// TwinCAT 3 PLC project plc_tmo_hutch_vac
// ProgramVersion: 3.1.4022.7
// libraries:
//   LCLS General, * (SLAC)
//   LCLS Vacuum, * (SLAC - LCLS)
//   LCLSVacuumSerialDriverLib, * (SLAC - LCLS)
//   PMPS, * (SLAC - LCLS)
//   Tc2_SerialCom, * (Beckhoff Automation GmbH)
//   Tc2_Standard, * (Beckhoff Automation GmbH)
//   Tc2_System, * (Beckhoff Automation GmbH)
//   Tc3_Module, * (Beckhoff Automation GmbH)
// project tree:
//   / ComTask.TcTTO, FSVTask.TcTTO, PlcTask.TcTTO
//   GVLs/ GVL_COM.TcGVL (not stored), GVL_FSV_PMPS.TcGVL (not stored), GVL_FS_Devices.TcGVL (not stored), GVL_Hutch_Gauges.TcGVL, GVL_Hutch_Pumps.TcGVL, GVL_Hutch_Valves.TcGVL, GVL_PMPS.TcGVL (not stored), GVL_Variables.TcGVL
//   POUs/ F_Turbo_Protection_ILK.TcPOU, MAIN.TcPOU, PMPS.TcPOU (not stored), PRG_COM.TcPOU (not stored), PRG_FEE.TcPOU, PRG_FSV.TcPOU (not stored), PRG_Hutch_Beamline_Valves.TcPOU, PRG_Hutch_Gauges.TcPOU, PRG_Roughing_Pumps.TcPOU
// real-time tasks:
//   TASK PlcTask: cycle T#10ms, priority 20, ADS port 350
//   TASK ComTask: cycle T#12ms, priority 21, ADS port 351
//   TASK FSVTask: cycle T#2ms, priority 19, ADS port 352
// I/O:
//   DEVICE Device 1 (EtherCAT), AmsNetId 172.21.132.45.2.1
//     Term 1 (EK1200)
//     TMO_WALL_WEST_EP01 (EP4374-0002)
//     TMO_K4S2_DRL_01 (EK1100) [EK1100 EtherCAT Coupler (2A E-Bus)]
//       K4S2_01_E1_VFS (EL1004)
//       K4S2_01_E2 (EL9190) [EL9190 Power Supplier]
//       K4S2_01_E3_VFS (EL2202)
//       K4S2_01_E4_VFS (EL2202)
//       K4S2_01_E5 (EL1004)
//       K4S2_01_E6 (EL2004)
//       Term 31 (EL9011)
//     TMO_K4S2_DRL_02 (EK1100) [EK1100 EtherCAT Coupler (2A E-Bus)]
//       K4S2_02_E1 (EL3174)
//       K4S2_02_E2 (EL3174)
//       K4S2_02_E3 (EL9184)
//       K4S2_02_E4 (EL9070) [EL9070 Shield terminal]
//       K4S2_02_E5 (EL2624)
//       K4S2_02_E6 (EL9505)
//       K4S2_02_E7 (EL1124) [EL1124 4Ch. Dig. Input 5V, 10µs, Sensor Power]
//       K4S2_02_E8 (EL1124)
//       K4S2_02_E9 (EL9410)
//       K4S2_02_E10 (EL6021) [EL6021 Interface (RS422/485)]
//       K4S2_02_E11 (EL1004)
//       K4S2_02_E12 (EL2794)
//       K4S2_02_E13 (EL1004)
//       K4S2_02_E14 (EL2794)
//       K4S2_02_E15 (EL1004)
//       K4S2_02_E16 (EL2794)
//       K4S2_02_E17 (EL6001) [EL6001 Interface (RS232)]
//       K4S2_02_E18 (EL6001) [EL6001 Interface (RS232)]
//       K4S2_02_E19 (EL1004)
//       K4S2_02_E20 (EL2004)
//       Term 32 (EL9011)
//     TMO_K4S2_ EP1 (EP4374-0002) [EP4374-0002 2Ch. Ana. Input +/-10V, 0-10V, 0/4-20mA configurable; 2Ch. Ana. Output +/-10V, 0-10V, 0/4-20mA configurable]
//     TMO_K4S6_ EP1 (EP4374-0002) [EP4374-0002 2Ch. Ana. Input +/-10V, 0-10V, 0/4-20mA configurable; 2Ch. Ana. Output +/-10V, 0-10V, 0/4-20mA configurable]
//     TMO_K4S6_DRL_01 (EK1100) [EK1100 EtherCAT Coupler (2A E-Bus)]
//       K4S6_01_E1 (EL1004)
//       K4S6_01_E2 (EL2004)
//       K4S6_01_E3 (EL1004)
//       K4S6_01_E4 (EL2004)
//       K4S6_01_E5 (EL6021) [EL6021 Schnittstelle (RS422/485)]
//       K4S6_01_E6 (EL1004)
//       K4S6_01_E7 (EL2004)
//       K4S6_01_E8 (EL1004)
//       K4S6_01_E9 (EL2004)
//       K4S6_01_E10 (EL6021)
//       K4S6_01_E11 (EL1004)
//       K4S6_01_E12 (EL2004)
//       K4S6_01_E13 (EL9410)
//       K4S6_01_E14 (EL2624)
//       K4S6_01_E15 (EL3174)
//       K4S6_01_E16 (EL9184) [EL9184 Potential Connection, 8 x 24V, 8 x Ground]
//       K4S6_01_E17 (EL9070) [EL9070 Shield terminal]
//       K4S6_01_E18 (EL3174)
//       K4S6_01_E19 (EL9505)
//       K4S6_01_E20 (EL1124)
//       K4S6_01_E21 (EL1124)
//       Term 119 (EL9410)
//       K4S6_01_E22_IP1 (EL1004)
//       K4S6_01_E23_IP1 (EL2794)
//       Term 91 (EL9011)
//     TMO_K4S8_DRL_01 (EK1100) [EK1100 EtherCAT Coupler (2A E-Bus)]
//       K4S8_01_E1 (EL1004)
//       K4S8_01_E2 (EL9190) [EL9190 Power Supplier]
//       K4S8_01_E3 (EL2202)
//       K4S8_01_E4 (EL2202)
//       K4S8_01_E5 (EL1004)
//       K4S8_01_E6 (EL2004)
//       Term 92 (EL9011)
// variable links:
//   plc_tmo_hutch_vac_fs/plc_tmo_hutch_vac_fs Instance <-> Device 1 (EtherCAT)/TMO_K4S2_DRL_01 (EK1100)/K4S2_01_E1_VFS (EL1004)
//     PlcTask Inputs/GVL_FS_Devices.MR3K4_KBO_VFS_1.i_xClsLS <-> Channel 1/Input
//     PlcTask Inputs/GVL_FS_Devices.MR3K4_KBO_VFS_1.i_xOpnLS <-> Channel 2/Input
//   plc_tmo_hutch_vac_fs/plc_tmo_hutch_vac_fs Instance <-> Device 1 (EtherCAT)/TMO_K4S2_DRL_01 (EK1100)/K4S2_01_E3_VFS (EL2202)
//     PlcTask Outputs/GVL_FS_Devices.MR3K4_KBO_VFS_1.q_xClose_A <-> Channel 1/Output
//     PlcTask Outputs/GVL_FS_Devices.MR3K4_KBO_VFS_1.q_xClose_B <-> Channel 2/Output
//   plc_tmo_hutch_vac_fs/plc_tmo_hutch_vac_fs Instance <-> Device 1 (EtherCAT)/TMO_K4S2_DRL_01 (EK1100)/K4S2_01_E4_VFS (EL2202)
//     PlcTask Outputs/GVL_FS_Devices.MR3K4_KBO_VFS_1.q_xClose_C <-> Channel 1/Output
//     PlcTask Outputs/GVL_FS_Devices.MR3K4_KBO_VFS_1.q_xOPN_DO <-> Channel 2/Output
//   plc_tmo_hutch_vac_fs/plc_tmo_hutch_vac_fs Instance <-> Device 1 (EtherCAT)/TMO_K4S8_DRL_01 (EK1100)/K4S8_01_E1 (EL1004)
//     PlcTask Inputs/GVL_FS_Devices.MR4K4_KBO_VFS_1.i_xClsLS <-> Channel 1/Input
//     PlcTask Inputs/GVL_FS_Devices.MR4K4_KBO_VFS_1.i_xOpnLS <-> Channel 2/Input
//   plc_tmo_hutch_vac_fs/plc_tmo_hutch_vac_fs Instance <-> Device 1 (EtherCAT)/TMO_K4S8_DRL_01 (EK1100)/K4S8_01_E3 (EL2202)
//     PlcTask Outputs/GVL_FS_Devices.MR4K4_KBO_VFS_1.q_xClose_A <-> Channel 1/Output
//     PlcTask Outputs/GVL_FS_Devices.MR4K4_KBO_VFS_1.q_xClose_B <-> Channel 2/Output
//   plc_tmo_hutch_vac_fs/plc_tmo_hutch_vac_fs Instance <-> Device 1 (EtherCAT)/TMO_K4S8_DRL_01 (EK1100)/K4S8_01_E4 (EL2202)
//     PlcTask Outputs/GVL_FS_Devices.MR4K4_KBO_VFS_1.q_xClose_C <-> Channel 1/Output
//     PlcTask Outputs/GVL_FS_Devices.MR4K4_KBO_VFS_1.q_xOPN_DO <-> Channel 2/Output
//   plc_tmo_hutch_vac Instance <-> Device 1 (EtherCAT)/TMO_K4S2_ EP1 (EP4374-0002)
//     ComTask Outputs/GVL_Hutch_Valves.TMO_ROUGH1_VFV_02.q_iRawPosition <-> AO Outputs Channel 3/Analog output
//     ComTask Outputs/GVL_Hutch_Valves.TMO_ROUGH2_VFV_01.q_iRawPosition <-> AO Outputs Channel 4/Analog output
//     PlcTask Inputs/GVL_Hutch_Gauges.TMO_ROUGH1_GPI_02.i_iPRESS_R <-> AI Inputs Channel 1/Value
//     PlcTask Inputs/GVL_Hutch_Gauges.TMO_ROUGH2_GPI_02.i_iPRESS_R <-> AI Inputs Channel 2/Value
//   plc_tmo_hutch_vac Instance <-> Device 1 (EtherCAT)/TMO_K4S2_DRL_01 (EK1100)/K4S2_01_E1_VFS (EL1004)
//     FSVTask Inputs/GVL_FS_Devices.MR3K4_KBO_VFS_1.i_xClsLS <-> Channel 1/Input
//     FSVTask Inputs/GVL_FS_Devices.MR3K4_KBO_VFS_1.i_xOpnLS <-> Channel 2/Input
//   plc_tmo_hutch_vac Instance <-> Device 1 (EtherCAT)/TMO_K4S2_DRL_01 (EK1100)/K4S2_01_E3_VFS (EL2202)
//     FSVTask Outputs/GVL_FS_Devices.MR3K4_KBO_VFS_1.q_xClose_A <-> Channel 1/Output
//     FSVTask Outputs/GVL_FS_Devices.MR3K4_KBO_VFS_1.q_xClose_B <-> Channel 2/Output
//   plc_tmo_hutch_vac Instance <-> Device 1 (EtherCAT)/TMO_K4S2_DRL_01 (EK1100)/K4S2_01_E4_VFS (EL2202)
//     FSVTask Outputs/GVL_FS_Devices.MR3K4_KBO_VFS_1.q_xClose_C <-> Channel 1/Output
//     FSVTask Outputs/GVL_FS_Devices.MR3K4_KBO_VFS_1.q_xOPN_DO <-> Channel 2/Output
//   plc_tmo_hutch_vac Instance <-> Device 1 (EtherCAT)/TMO_K4S2_DRL_01 (EK1100)/K4S2_01_E5 (EL1004)
//     PlcTask Inputs/GVL_Hutch_Valves.MR2K4_KBO_VWC_01.i_xClsLS <-> Channel 2/Input
//     PlcTask Inputs/GVL_Hutch_Valves.MR3K4_KBO_VWC_01.i_xClsLS <-> Channel 4/Input
//     PlcTask Inputs/GVL_Hutch_Valves.MR2K4_KBO_VWC_01.i_xOpnLS <-> Channel 1/Input
//     PlcTask Inputs/GVL_Hutch_Valves.MR3K4_KBO_VWC_01.i_xOpnLS <-> Channel 3/Input
//   plc_tmo_hutch_vac Instance <-> Device 1 (EtherCAT)/TMO_K4S2_DRL_01 (EK1100)/K4S2_01_E6 (EL2004)
//     PlcTask Outputs/GVL_Hutch_Valves.MR2K4_KBO_VWC_01.q_xOPN_DO <-> Channel 1/Output
//     PlcTask Outputs/GVL_Hutch_Valves.MR3K4_KBO_VWC_01.q_xOPN_DO <-> Channel 2/Output
//   plc_tmo_hutch_vac Instance <-> Device 1 (EtherCAT)/TMO_K4S2_DRL_02 (EK1100)/K4S2_02_E1 (EL3174)
//     PlcTask Inputs/GVL_Hutch_Gauges.MR2K4_KBO_GCC_01.i_iPRESS_R <-> AI Standard Channel 3/Value
//     PlcTask Inputs/GVL_Hutch_Gauges.MR2K4_KBO_GPI_01.i_iPRESS_R <-> AI Standard Channel 2/Value
//     PlcTask Inputs/GVL_Hutch_Gauges.PA1K4_IP1_GCC_01.i_iPRESS_R <-> AI Standard Channel 4/Value
//   plc_tmo_hutch_vac Instance <-> Device 1 (EtherCAT)/TMO_K4S2_DRL_02 (EK1100)/K4S2_02_E10 (EL6021)
//     ComTask Inputs/GVL_COM.K4S2_02_E10_stComIn/D[0] <-> COM TxPDO-Map Inputs/Data In 0
//     ComTask Inputs/GVL_COM.K4S2_02_E10_stComIn/D[10] <-> COM TxPDO-Map Inputs/Data In 10
//     ComTask Inputs/GVL_COM.K4S2_02_E10_stComIn/D[11] <-> COM TxPDO-Map Inputs/Data In 11
//     ComTask Inputs/GVL_COM.K4S2_02_E10_stComIn/D[12] <-> COM TxPDO-Map Inputs/Data In 12
//     ComTask Inputs/GVL_COM.K4S2_02_E10_stComIn/D[13] <-> COM TxPDO-Map Inputs/Data In 13
//     ComTask Inputs/GVL_COM.K4S2_02_E10_stComIn/D[14] <-> COM TxPDO-Map Inputs/Data In 14
//     ComTask Inputs/GVL_COM.K4S2_02_E10_stComIn/D[15] <-> COM TxPDO-Map Inputs/Data In 15
//     ComTask Inputs/GVL_COM.K4S2_02_E10_stComIn/D[16] <-> COM TxPDO-Map Inputs/Data In 16
//     ComTask Inputs/GVL_COM.K4S2_02_E10_stComIn/D[17] <-> COM TxPDO-Map Inputs/Data In 17
//     ComTask Inputs/GVL_COM.K4S2_02_E10_stComIn/D[18] <-> COM TxPDO-Map Inputs/Data In 18
//     ComTask Inputs/GVL_COM.K4S2_02_E10_stComIn/D[19] <-> COM TxPDO-Map Inputs/Data In 19
//     ComTask Inputs/GVL_COM.K4S2_02_E10_stComIn/D[1] <-> COM TxPDO-Map Inputs/Data In 1
//     ComTask Inputs/GVL_COM.K4S2_02_E10_stComIn/D[20] <-> COM TxPDO-Map Inputs/Data In 20
//     ComTask Inputs/GVL_COM.K4S2_02_E10_stComIn/D[21] <-> COM TxPDO-Map Inputs/Data In 21
//     ComTask Inputs/GVL_COM.K4S2_02_E10_stComIn/D[2] <-> COM TxPDO-Map Inputs/Data In 2
//     ComTask Inputs/GVL_COM.K4S2_02_E10_stComIn/D[3] <-> COM TxPDO-Map Inputs/Data In 3
//     ComTask Inputs/GVL_COM.K4S2_02_E10_stComIn/D[4] <-> COM TxPDO-Map Inputs/Data In 4
//     ComTask Inputs/GVL_COM.K4S2_02_E10_stComIn/D[5] <-> COM TxPDO-Map Inputs/Data In 5
//     ComTask Inputs/GVL_COM.K4S2_02_E10_stComIn/D[6] <-> COM TxPDO-Map Inputs/Data In 6
//     ComTask Inputs/GVL_COM.K4S2_02_E10_stComIn/D[7] <-> COM TxPDO-Map Inputs/Data In 7
//     ComTask Inputs/GVL_COM.K4S2_02_E10_stComIn/D[8] <-> COM TxPDO-Map Inputs/Data In 8
//     ComTask Inputs/GVL_COM.K4S2_02_E10_stComIn/D[9] <-> COM TxPDO-Map Inputs/Data In 9
//     ComTask Inputs/GVL_COM.K4S2_02_E10_stComIn/Status <-> COM TxPDO-Map Inputs/Status
//     ComTask Outputs/GVL_COM.K4S2_02_E10_stComOut/Ctrl <-> COM RxPDO-Map Outputs/Ctrl
//     ComTask Outputs/GVL_COM.K4S2_02_E10_stComOut/D[0] <-> COM RxPDO-Map Outputs/Data Out 0
//     ComTask Outputs/GVL_COM.K4S2_02_E10_stComOut/D[10] <-> COM RxPDO-Map Outputs/Data Out 10
//     ComTask Outputs/GVL_COM.K4S2_02_E10_stComOut/D[11] <-> COM RxPDO-Map Outputs/Data Out 11
//     ComTask Outputs/GVL_COM.K4S2_02_E10_stComOut/D[12] <-> COM RxPDO-Map Outputs/Data Out 12
//     ComTask Outputs/GVL_COM.K4S2_02_E10_stComOut/D[13] <-> COM RxPDO-Map Outputs/Data Out 13
//     ComTask Outputs/GVL_COM.K4S2_02_E10_stComOut/D[14] <-> COM RxPDO-Map Outputs/Data Out 14
//     ComTask Outputs/GVL_COM.K4S2_02_E10_stComOut/D[15] <-> COM RxPDO-Map Outputs/Data Out 15
//     ComTask Outputs/GVL_COM.K4S2_02_E10_stComOut/D[16] <-> COM RxPDO-Map Outputs/Data Out 16
//     ComTask Outputs/GVL_COM.K4S2_02_E10_stComOut/D[17] <-> COM RxPDO-Map Outputs/Data Out 17
//     ComTask Outputs/GVL_COM.K4S2_02_E10_stComOut/D[18] <-> COM RxPDO-Map Outputs/Data Out 18
//     ComTask Outputs/GVL_COM.K4S2_02_E10_stComOut/D[19] <-> COM RxPDO-Map Outputs/Data Out 19
//     ComTask Outputs/GVL_COM.K4S2_02_E10_stComOut/D[1] <-> COM RxPDO-Map Outputs/Data Out 1
//     ComTask Outputs/GVL_COM.K4S2_02_E10_stComOut/D[20] <-> COM RxPDO-Map Outputs/Data Out 20
//     ComTask Outputs/GVL_COM.K4S2_02_E10_stComOut/D[21] <-> COM RxPDO-Map Outputs/Data Out 21
//     ComTask Outputs/GVL_COM.K4S2_02_E10_stComOut/D[2] <-> COM RxPDO-Map Outputs/Data Out 2
//     ComTask Outputs/GVL_COM.K4S2_02_E10_stComOut/D[3] <-> COM RxPDO-Map Outputs/Data Out 3
//     ComTask Outputs/GVL_COM.K4S2_02_E10_stComOut/D[4] <-> COM RxPDO-Map Outputs/Data Out 4
//     ComTask Outputs/GVL_COM.K4S2_02_E10_stComOut/D[5] <-> COM RxPDO-Map Outputs/Data Out 5
//     ComTask Outputs/GVL_COM.K4S2_02_E10_stComOut/D[6] <-> COM RxPDO-Map Outputs/Data Out 6
//     ComTask Outputs/GVL_COM.K4S2_02_E10_stComOut/D[7] <-> COM RxPDO-Map Outputs/Data Out 7
//     ComTask Outputs/GVL_COM.K4S2_02_E10_stComOut/D[8] <-> COM RxPDO-Map Outputs/Data Out 8
//     ComTask Outputs/GVL_COM.K4S2_02_E10_stComOut/D[9] <-> COM RxPDO-Map Outputs/Data Out 9
//   plc_tmo_hutch_vac Instance <-> Device 1 (EtherCAT)/TMO_K4S2_DRL_02 (EK1100)/K4S2_02_E11 (EL1004)
//     PlcTask Inputs/GVL_Hutch_Pumps.PA1K4_IP1_PTM_01.i_xAtSpd <-> Channel 2/Input
//     PlcTask Inputs/GVL_Hutch_Pumps.PA1K4_IP1_PTM_02.i_xAtSpd <-> Channel 4/Input
//     PlcTask Inputs/GVL_Hutch_Pumps.PA1K4_IP1_PTM_01.i_xFaultNC <-> Channel 1/Input
//     PlcTask Inputs/GVL_Hutch_Pumps.PA1K4_IP1_PTM_02.i_xFaultNC <-> Channel 3/Input
//   plc_tmo_hutch_vac Instance <-> Device 1 (EtherCAT)/TMO_K4S2_DRL_02 (EK1100)/K4S2_02_E12 (EL2794)
//     PlcTask Outputs/GVL_Hutch_Pumps.PA1K4_IP1_PTM_01.q_RunDO <-> Channel 1/Output
//     PlcTask Outputs/GVL_Hutch_Pumps.PA1K4_IP1_PTM_02.q_RunDO <-> Channel 3/Output
//     PlcTask Outputs/GVL_Hutch_Pumps.PA1K4_IP1_PTM_01.q_xReset <-> Channel 2/Output
//     PlcTask Outputs/GVL_Hutch_Pumps.PA1K4_IP1_PTM_02.q_xReset <-> Channel 4/Output
//   plc_tmo_hutch_vac Instance <-> Device 1 (EtherCAT)/TMO_K4S2_DRL_02 (EK1100)/K4S2_02_E13 (EL1004)
//     PlcTask Inputs/GVL_Hutch_Pumps.PA1K4_IP1_PTM_03.i_xAtSpd <-> Channel 2/Input
//     PlcTask Inputs/GVL_Hutch_Pumps.PA1K4_IP1_PTM_03.i_xFaultNC <-> Channel 1/Input
//   plc_tmo_hutch_vac Instance <-> Device 1 (EtherCAT)/TMO_K4S2_DRL_02 (EK1100)/K4S2_02_E14 (EL2794)
//     PlcTask Outputs/GVL_Hutch_Pumps.PA1K4_IP1_PTM_03.q_RunDO <-> Channel 1/Output
//     PlcTask Outputs/GVL_Hutch_Pumps.PA1K4_IP1_PTM_03.q_xReset <-> Channel 2/Output
//   plc_tmo_hutch_vac Instance <-> Device 1 (EtherCAT)/TMO_K4S2_DRL_02 (EK1100)/K4S2_02_E15 (EL1004)
//     PlcTask Inputs/GVL_Hutch_Pumps.IM4K4_PPM_PTM_01.i_xAtSpd <-> Channel 2/Input
//     PlcTask Inputs/GVL_Hutch_Pumps.IM4K4_PPM_PTM_01.i_xFaultNC <-> Channel 1/Input
//     PlcTask Inputs/GVL_Hutch_Pumps.LI1K4_IP1_PTM_01.i_xAtSpd <-> Channel 4/Input
//     PlcTask Inputs/GVL_Hutch_Pumps.LI1K4_IP1_PTM_01.i_xFaultNC <-> Channel 3/Input
//   plc_tmo_hutch_vac Instance <-> Device 1 (EtherCAT)/TMO_K4S2_DRL_02 (EK1100)/K4S2_02_E16 (EL2794)
//     PlcTask Outputs/GVL_Hutch_Pumps.IM4K4_PPM_PTM_01.q_RunDO <-> Channel 1/Output
//     PlcTask Outputs/GVL_Hutch_Pumps.LI1K4_IP1_PTM_01.q_RunDO <-> Channel 2/Output
//   plc_tmo_hutch_vac Instance <-> Device 1 (EtherCAT)/TMO_K4S2_DRL_02 (EK1100)/K4S2_02_E17 (EL6001)
//     ComTask Inputs/GVL_COM.K4S2_02_E17_stComIn/D[0] <-> COM Inputs/Data In 0
//     ComTask Inputs/GVL_COM.K4S2_02_E17_stComIn/D[10] <-> COM Inputs/Data In 10
//     ComTask Inputs/GVL_COM.K4S2_02_E17_stComIn/D[11] <-> COM Inputs/Data In 11
//     ComTask Inputs/GVL_COM.K4S2_02_E17_stComIn/D[12] <-> COM Inputs/Data In 12
//     ComTask Inputs/GVL_COM.K4S2_02_E17_stComIn/D[13] <-> COM Inputs/Data In 13
//     ComTask Inputs/GVL_COM.K4S2_02_E17_stComIn/D[14] <-> COM Inputs/Data In 14
//     ComTask Inputs/GVL_COM.K4S2_02_E17_stComIn/D[15] <-> COM Inputs/Data In 15
//     ComTask Inputs/GVL_COM.K4S2_02_E17_stComIn/D[16] <-> COM Inputs/Data In 16
//     ComTask Inputs/GVL_COM.K4S2_02_E17_stComIn/D[17] <-> COM Inputs/Data In 17
//     ComTask Inputs/GVL_COM.K4S2_02_E17_stComIn/D[18] <-> COM Inputs/Data In 18
//     ComTask Inputs/GVL_COM.K4S2_02_E17_stComIn/D[19] <-> COM Inputs/Data In 19
//     ComTask Inputs/GVL_COM.K4S2_02_E17_stComIn/D[1] <-> COM Inputs/Data In 1
//     ComTask Inputs/GVL_COM.K4S2_02_E17_stComIn/D[20] <-> COM Inputs/Data In 20
//     ComTask Inputs/GVL_COM.K4S2_02_E17_stComIn/D[21] <-> COM Inputs/Data In 21
//     ComTask Inputs/GVL_COM.K4S2_02_E17_stComIn/D[2] <-> COM Inputs/Data In 2
//     ComTask Inputs/GVL_COM.K4S2_02_E17_stComIn/D[3] <-> COM Inputs/Data In 3
//     ComTask Inputs/GVL_COM.K4S2_02_E17_stComIn/D[4] <-> COM Inputs/Data In 4
//     ComTask Inputs/GVL_COM.K4S2_02_E17_stComIn/D[5] <-> COM Inputs/Data In 5
//     ComTask Inputs/GVL_COM.K4S2_02_E17_stComIn/D[6] <-> COM Inputs/Data In 6
//     ComTask Inputs/GVL_COM.K4S2_02_E17_stComIn/D[7] <-> COM Inputs/Data In 7
//     ComTask Inputs/GVL_COM.K4S2_02_E17_stComIn/D[8] <-> COM Inputs/Data In 8
//     ComTask Inputs/GVL_COM.K4S2_02_E17_stComIn/D[9] <-> COM Inputs/Data In 9
//     ComTask Inputs/GVL_COM.K4S2_02_E17_stComIn/Status <-> COM Inputs/Status
//     ComTask Outputs/GVL_COM.K4S2_02_E17_stComOut/Ctrl <-> COM Outputs/Ctrl
//     ComTask Outputs/GVL_COM.K4S2_02_E17_stComOut/D[0] <-> COM Outputs/Data Out 0
//     ComTask Outputs/GVL_COM.K4S2_02_E17_stComOut/D[10] <-> COM Outputs/Data Out 10
//     ComTask Outputs/GVL_COM.K4S2_02_E17_stComOut/D[11] <-> COM Outputs/Data Out 11
//     ComTask Outputs/GVL_COM.K4S2_02_E17_stComOut/D[12] <-> COM Outputs/Data Out 12
//     ComTask Outputs/GVL_COM.K4S2_02_E17_stComOut/D[13] <-> COM Outputs/Data Out 13
//     ComTask Outputs/GVL_COM.K4S2_02_E17_stComOut/D[14] <-> COM Outputs/Data Out 14
//     ComTask Outputs/GVL_COM.K4S2_02_E17_stComOut/D[15] <-> COM Outputs/Data Out 15
//     ComTask Outputs/GVL_COM.K4S2_02_E17_stComOut/D[16] <-> COM Outputs/Data Out 16
//     ComTask Outputs/GVL_COM.K4S2_02_E17_stComOut/D[17] <-> COM Outputs/Data Out 17
//     ComTask Outputs/GVL_COM.K4S2_02_E17_stComOut/D[18] <-> COM Outputs/Data Out 18
//     ComTask Outputs/GVL_COM.K4S2_02_E17_stComOut/D[19] <-> COM Outputs/Data Out 19
//     ComTask Outputs/GVL_COM.K4S2_02_E17_stComOut/D[1] <-> COM Outputs/Data Out 1
//     ComTask Outputs/GVL_COM.K4S2_02_E17_stComOut/D[20] <-> COM Outputs/Data Out 20
//     ComTask Outputs/GVL_COM.K4S2_02_E17_stComOut/D[21] <-> COM Outputs/Data Out 21
//     ComTask Outputs/GVL_COM.K4S2_02_E17_stComOut/D[2] <-> COM Outputs/Data Out 2
//     ComTask Outputs/GVL_COM.K4S2_02_E17_stComOut/D[3] <-> COM Outputs/Data Out 3
//     ComTask Outputs/GVL_COM.K4S2_02_E17_stComOut/D[4] <-> COM Outputs/Data Out 4
//     ComTask Outputs/GVL_COM.K4S2_02_E17_stComOut/D[5] <-> COM Outputs/Data Out 5
//     ComTask Outputs/GVL_COM.K4S2_02_E17_stComOut/D[6] <-> COM Outputs/Data Out 6
//     ComTask Outputs/GVL_COM.K4S2_02_E17_stComOut/D[7] <-> COM Outputs/Data Out 7
//     ComTask Outputs/GVL_COM.K4S2_02_E17_stComOut/D[8] <-> COM Outputs/Data Out 8
//     ComTask Outputs/GVL_COM.K4S2_02_E17_stComOut/D[9] <-> COM Outputs/Data Out 9
//   plc_tmo_hutch_vac Instance <-> Device 1 (EtherCAT)/TMO_K4S2_DRL_02 (EK1100)/K4S2_02_E18 (EL6001)
//     ComTask Inputs/GVL_COM.K4S2_02_E18_stComIn/D[0] <-> COM Inputs/Data In 0
//     ComTask Inputs/GVL_COM.K4S2_02_E18_stComIn/D[10] <-> COM Inputs/Data In 10
//     ComTask Inputs/GVL_COM.K4S2_02_E18_stComIn/D[11] <-> COM Inputs/Data In 11
//     ComTask Inputs/GVL_COM.K4S2_02_E18_stComIn/D[12] <-> COM Inputs/Data In 12
//     ComTask Inputs/GVL_COM.K4S2_02_E18_stComIn/D[13] <-> COM Inputs/Data In 13
//     ComTask Inputs/GVL_COM.K4S2_02_E18_stComIn/D[14] <-> COM Inputs/Data In 14
//     ComTask Inputs/GVL_COM.K4S2_02_E18_stComIn/D[15] <-> COM Inputs/Data In 15
//     ComTask Inputs/GVL_COM.K4S2_02_E18_stComIn/D[16] <-> COM Inputs/Data In 16
//     ComTask Inputs/GVL_COM.K4S2_02_E18_stComIn/D[17] <-> COM Inputs/Data In 17
//     ComTask Inputs/GVL_COM.K4S2_02_E18_stComIn/D[18] <-> COM Inputs/Data In 18
//     ComTask Inputs/GVL_COM.K4S2_02_E18_stComIn/D[19] <-> COM Inputs/Data In 19
//     ComTask Inputs/GVL_COM.K4S2_02_E18_stComIn/D[1] <-> COM Inputs/Data In 1
//     ComTask Inputs/GVL_COM.K4S2_02_E18_stComIn/D[20] <-> COM Inputs/Data In 20
//     ComTask Inputs/GVL_COM.K4S2_02_E18_stComIn/D[21] <-> COM Inputs/Data In 21
//     ComTask Inputs/GVL_COM.K4S2_02_E18_stComIn/D[2] <-> COM Inputs/Data In 2
//     ComTask Inputs/GVL_COM.K4S2_02_E18_stComIn/D[3] <-> COM Inputs/Data In 3
//     ComTask Inputs/GVL_COM.K4S2_02_E18_stComIn/D[4] <-> COM Inputs/Data In 4
//     ComTask Inputs/GVL_COM.K4S2_02_E18_stComIn/D[5] <-> COM Inputs/Data In 5
//     ComTask Inputs/GVL_COM.K4S2_02_E18_stComIn/D[6] <-> COM Inputs/Data In 6
//     ComTask Inputs/GVL_COM.K4S2_02_E18_stComIn/D[7] <-> COM Inputs/Data In 7
//     ComTask Inputs/GVL_COM.K4S2_02_E18_stComIn/D[8] <-> COM Inputs/Data In 8
//     ComTask Inputs/GVL_COM.K4S2_02_E18_stComIn/D[9] <-> COM Inputs/Data In 9
//     ComTask Inputs/GVL_COM.K4S2_02_E18_stComIn/Status <-> COM Inputs/Status
//     ComTask Outputs/GVL_COM.K4S2_02_E18_stComOut/Ctrl <-> COM Outputs/Ctrl
//     ComTask Outputs/GVL_COM.K4S2_02_E18_stComOut/D[0] <-> COM Outputs/Data Out 0
//     ComTask Outputs/GVL_COM.K4S2_02_E18_stComOut/D[10] <-> COM Outputs/Data Out 10
//     ComTask Outputs/GVL_COM.K4S2_02_E18_stComOut/D[11] <-> COM Outputs/Data Out 11
//     ComTask Outputs/GVL_COM.K4S2_02_E18_stComOut/D[12] <-> COM Outputs/Data Out 12
//     ComTask Outputs/GVL_COM.K4S2_02_E18_stComOut/D[13] <-> COM Outputs/Data Out 13
//     ComTask Outputs/GVL_COM.K4S2_02_E18_stComOut/D[14] <-> COM Outputs/Data Out 14
//     ComTask Outputs/GVL_COM.K4S2_02_E18_stComOut/D[15] <-> COM Outputs/Data Out 15
//     ComTask Outputs/GVL_COM.K4S2_02_E18_stComOut/D[16] <-> COM Outputs/Data Out 16
//     ComTask Outputs/GVL_COM.K4S2_02_E18_stComOut/D[17] <-> COM Outputs/Data Out 17
//     ComTask Outputs/GVL_COM.K4S2_02_E18_stComOut/D[18] <-> COM Outputs/Data Out 18
//     ComTask Outputs/GVL_COM.K4S2_02_E18_stComOut/D[19] <-> COM Outputs/Data Out 19
//     ComTask Outputs/GVL_COM.K4S2_02_E18_stComOut/D[1] <-> COM Outputs/Data Out 1
//     ComTask Outputs/GVL_COM.K4S2_02_E18_stComOut/D[20] <-> COM Outputs/Data Out 20
//     ComTask Outputs/GVL_COM.K4S2_02_E18_stComOut/D[21] <-> COM Outputs/Data Out 21
//     ComTask Outputs/GVL_COM.K4S2_02_E18_stComOut/D[2] <-> COM Outputs/Data Out 2
//     ComTask Outputs/GVL_COM.K4S2_02_E18_stComOut/D[3] <-> COM Outputs/Data Out 3
//     ComTask Outputs/GVL_COM.K4S2_02_E18_stComOut/D[4] <-> COM Outputs/Data Out 4
//     ComTask Outputs/GVL_COM.K4S2_02_E18_stComOut/D[5] <-> COM Outputs/Data Out 5
//     ComTask Outputs/GVL_COM.K4S2_02_E18_stComOut/D[6] <-> COM Outputs/Data Out 6
//     ComTask Outputs/GVL_COM.K4S2_02_E18_stComOut/D[7] <-> COM Outputs/Data Out 7
//     ComTask Outputs/GVL_COM.K4S2_02_E18_stComOut/D[8] <-> COM Outputs/Data Out 8
//     ComTask Outputs/GVL_COM.K4S2_02_E18_stComOut/D[9] <-> COM Outputs/Data Out 9
//   plc_tmo_hutch_vac Instance <-> Device 1 (EtherCAT)/TMO_K4S2_DRL_02 (EK1100)/K4S2_02_E19 (EL1004)
//     PlcTask Inputs/GVL_Hutch_Valves.TMO_ROUGH1_VRC_01.i_xClsLS <-> Channel 2/Input
//     PlcTask Inputs/GVL_Hutch_Valves.TMO_ROUGH2_VRC_01.i_xClsLS <-> Channel 4/Input
//     PlcTask Inputs/GVL_Hutch_Valves.TMO_ROUGH1_VRC_01.i_xOpnLS <-> Channel 1/Input
//     PlcTask Inputs/GVL_Hutch_Valves.TMO_ROUGH2_VRC_01.i_xOpnLS <-> Channel 3/Input
//   plc_tmo_hutch_vac Instance <-> Device 1 (EtherCAT)/TMO_K4S2_DRL_02 (EK1100)/K4S2_02_E2 (EL3174)
//     PlcTask Inputs/GVL_Hutch_Gauges.IM4K4_PPM_GCC_01.i_iPRESS_R <-> AI Standard Channel 2/Value
//     PlcTask Inputs/GVL_Hutch_Gauges.PA1K4_IP1_GPI_01.i_iPRESS_R <-> AI Standard Channel 1/Value
//   plc_tmo_hutch_vac Instance <-> Device 1 (EtherCAT)/TMO_K4S2_DRL_02 (EK1100)/K4S2_02_E20 (EL2004)
//     PlcTask Outputs/GVL_Hutch_Valves.TMO_ROUGH1_VRC_01.q_xOPN_DO <-> Channel 1/Output
//     PlcTask Outputs/GVL_Hutch_Valves.TMO_ROUGH2_VRC_01.q_xOPN_DO <-> Channel 2/Output
//   plc_tmo_hutch_vac Instance <-> Device 1 (EtherCAT)/TMO_K4S2_DRL_02 (EK1100)/K4S2_02_E5 (EL2624)
//     PlcTask Outputs/GVL_Hutch_Gauges.IM4K4_PPM_GCC_01.q_xHV_DIS <-> Channel 4/Output
//     PlcTask Outputs/GVL_Hutch_Gauges.MR2K4_KBO_GCC_01.q_xHV_DIS <-> Channel 2/Output
//     PlcTask Outputs/GVL_Hutch_Gauges.PA1K4_IP1_GCC_01.q_xHV_DIS <-> Channel 3/Output
//   plc_tmo_hutch_vac Instance <-> Device 1 (EtherCAT)/TMO_K4S2_DRL_02 (EK1100)/K4S2_02_E7 (EL1124)
//     PlcTask Inputs/GVL_Hutch_Gauges.MR2K4_KBO_GCC_01.i_xDisc_Active <-> Channel 4/Input
//     PlcTask Inputs/GVL_Hutch_Gauges.MR2K4_KBO_GCC_01.i_xHV_ON <-> Channel 3/Input
//   plc_tmo_hutch_vac Instance <-> Device 1 (EtherCAT)/TMO_K4S2_DRL_02 (EK1100)/K4S2_02_E8 (EL1124)
//     PlcTask Inputs/GVL_Hutch_Gauges.IM4K4_PPM_GCC_01.i_xDisc_Active <-> Channel 4/Input
//     PlcTask Inputs/GVL_Hutch_Gauges.IM4K4_PPM_GCC_01.i_xHV_ON <-> Channel 3/Input
//     PlcTask Inputs/GVL_Hutch_Gauges.PA1K4_IP1_GCC_01.i_xDisc_Active <-> Channel 2/Input
//     PlcTask Inputs/GVL_Hutch_Gauges.PA1K4_IP1_GCC_01.i_xHV_ON <-> Channel 1/Input
//   plc_tmo_hutch_vac Instance <-> Device 1 (EtherCAT)/TMO_K4S6_ EP1 (EP4374-0002)
//     ComTask Outputs/GVL_Hutch_Valves.TMO_ROUGH1_VFV_03.q_iRawPosition <-> AO Outputs Channel 3/Analog output
//     PlcTask Inputs/GVL_Hutch_Gauges.TMO_ROUGH1_GPI_03.i_iPRESS_R <-> AI Inputs Channel 1/Value
//   plc_tmo_hutch_vac Instance <-> Device 1 (EtherCAT)/TMO_K4S6_DRL_01 (EK1100)/K4S6_01_E1 (EL1004)
//     PlcTask Inputs/GVL_Hutch_Valves.TMO_ROUGH1_VRC_02.i_xClsLS <-> Channel 2/Input
//     PlcTask Inputs/GVL_Hutch_Valves.TMO_ROUGH1_VRC_02.i_xOpnLS <-> Channel 1/Input
//   plc_tmo_hutch_vac Instance <-> Device 1 (EtherCAT)/TMO_K4S6_DRL_01 (EK1100)/K4S6_01_E11 (EL1004)
//     PlcTask Inputs/GVL_Hutch_Pumps.IM5K4_PPM_PTM_01.i_xFaultNC <-> Channel 1/Input
//   plc_tmo_hutch_vac Instance <-> Device 1 (EtherCAT)/TMO_K4S6_DRL_01 (EK1100)/K4S6_01_E12 (EL2004)
//     PlcTask Outputs/GVL_Hutch_Pumps.IM5K4_PPM_PTM_01.q_PumpingStation <-> Channel 1/Output
//   plc_tmo_hutch_vac Instance <-> Device 1 (EtherCAT)/TMO_K4S6_DRL_01 (EK1100)/K4S6_01_E14 (EL2624)
//     PlcTask Outputs/GVL_Hutch_Gauges.IM5K4_PPM_GCC_01.q_xHV_DIS <-> Channel 2/Output
//     PlcTask Outputs/GVL_Hutch_Gauges.MR4K4_KBO_GCC_01.q_xHV_DIS <-> Channel 4/Output
//     PlcTask Outputs/GVL_Hutch_Gauges.PA2K4_IP1_GCC_01.q_xHV_DIS <-> Channel 3/Output
//     PlcTask Outputs/GVL_Hutch_Gauges.TM1K4_GCC_01.q_xHV_DIS <-> Channel 1/Output
//   plc_tmo_hutch_vac Instance <-> Device 1 (EtherCAT)/TMO_K4S6_DRL_01 (EK1100)/K4S6_01_E15 (EL3174)
//     PlcTask Inputs/GVL_Hutch_Gauges.IM5K4_PPM_GCC_01.i_iPRESS_R <-> AI Standard Channel 2/Value
//     PlcTask Inputs/GVL_Hutch_Gauges.PA2K4_IP1_GCC_01.i_iPRESS_R <-> AI Standard Channel 3/Value
//     PlcTask Inputs/GVL_Hutch_Gauges.PA2K4_IP1_GPI_01.i_iPRESS_R <-> AI Standard Channel 4/Value
//     PlcTask Inputs/GVL_Hutch_Gauges.TM1K4_GCC_01.i_iPRESS_R <-> AI Standard Channel 1/Value
//   plc_tmo_hutch_vac Instance <-> Device 1 (EtherCAT)/TMO_K4S6_DRL_01 (EK1100)/K4S6_01_E18 (EL3174)
//     PlcTask Inputs/GVL_Hutch_Gauges.MR4K4_KBO_GCC_01.i_iPRESS_R <-> AI Standard Channel 2/Value
//     PlcTask Inputs/GVL_Hutch_Gauges.MR4K4_KBO_GPI_01.i_iPRESS_R <-> AI Standard Channel 1/Value
//   plc_tmo_hutch_vac Instance <-> Device 1 (EtherCAT)/TMO_K4S6_DRL_01 (EK1100)/K4S6_01_E2 (EL2004)
//     PlcTask Outputs/GVL_Hutch_Valves.TMO_ROUGH1_VRC_02.q_xOPN_DO <-> Channel 1/Output
//   plc_tmo_hutch_vac Instance <-> Device 1 (EtherCAT)/TMO_K4S6_DRL_01 (EK1100)/K4S6_01_E20 (EL1124)
//     PlcTask Inputs/GVL_Hutch_Gauges.IM5K4_PPM_GCC_01.i_xDisc_Active <-> Channel 4/Input
//     PlcTask Inputs/GVL_Hutch_Gauges.IM5K4_PPM_GCC_01.i_xHV_ON <-> Channel 3/Input
//     PlcTask Inputs/GVL_Hutch_Gauges.TM1K4_GCC_01.i_xDisc_Active <-> Channel 2/Input
//     PlcTask Inputs/GVL_Hutch_Gauges.TM1K4_GCC_01.i_xHV_ON <-> Channel 1/Input
//   plc_tmo_hutch_vac Instance <-> Device 1 (EtherCAT)/TMO_K4S6_DRL_01 (EK1100)/K4S6_01_E21 (EL1124)
//     PlcTask Inputs/GVL_Hutch_Gauges.MR4K4_KBO_GCC_01.i_xDisc_Active <-> Channel 4/Input
//     PlcTask Inputs/GVL_Hutch_Gauges.MR4K4_KBO_GCC_01.i_xHV_ON <-> Channel 3/Input
//     PlcTask Inputs/GVL_Hutch_Gauges.PA2K4_IP1_GCC_01.i_xDisc_Active <-> Channel 2/Input
//     PlcTask Inputs/GVL_Hutch_Gauges.PA2K4_IP1_GCC_01.i_xHV_ON <-> Channel 1/Input
//   plc_tmo_hutch_vac Instance <-> Device 1 (EtherCAT)/TMO_K4S6_DRL_01 (EK1100)/K4S6_01_E3 (EL1004)
//     PlcTask Inputs/GVL_Hutch_Valves.LI3K4_IP1_VWC_01.i_xClsLS <-> Channel 2/Input
//     PlcTask Inputs/GVL_Hutch_Valves.LI3K4_IP1_VWC_01.i_xOpnLS <-> Channel 1/Input
//     PlcTask Inputs/GVL_Hutch_Valves.PC5K4_VWC_01.i_xClsLS <-> Channel 4/Input
//     PlcTask Inputs/GVL_Hutch_Valves.PC5K4_VWC_01.i_xOpnLS <-> Channel 3/Input
//   plc_tmo_hutch_vac Instance <-> Device 1 (EtherCAT)/TMO_K4S6_DRL_01 (EK1100)/K4S6_01_E4 (EL2004)
//     PlcTask Outputs/GVL_Hutch_Valves.LI3K4_IP1_VWC_01.q_xOPN_DO <-> Channel 1/Output
//     PlcTask Outputs/GVL_Hutch_Valves.PC5K4_VWC_01.q_xOPN_DO <-> Channel 2/Output
//   plc_tmo_hutch_vac Instance <-> Device 1 (EtherCAT)/TMO_K4S6_DRL_01 (EK1100)/K4S6_01_E5 (EL6021)
//     ComTask Inputs/GVL_COM.K4S6_01_E5_stComIn/D[0] <-> COM TxPDO-Map Inputs/Data In 0
//     ComTask Inputs/GVL_COM.K4S6_01_E5_stComIn/D[10] <-> COM TxPDO-Map Inputs/Data In 10
//     ComTask Inputs/GVL_COM.K4S6_01_E5_stComIn/D[11] <-> COM TxPDO-Map Inputs/Data In 11
//     ComTask Inputs/GVL_COM.K4S6_01_E5_stComIn/D[12] <-> COM TxPDO-Map Inputs/Data In 12
//     ComTask Inputs/GVL_COM.K4S6_01_E5_stComIn/D[13] <-> COM TxPDO-Map Inputs/Data In 13
//     ComTask Inputs/GVL_COM.K4S6_01_E5_stComIn/D[14] <-> COM TxPDO-Map Inputs/Data In 14
//     ComTask Inputs/GVL_COM.K4S6_01_E5_stComIn/D[15] <-> COM TxPDO-Map Inputs/Data In 15
//     ComTask Inputs/GVL_COM.K4S6_01_E5_stComIn/D[16] <-> COM TxPDO-Map Inputs/Data In 16
//     ComTask Inputs/GVL_COM.K4S6_01_E5_stComIn/D[17] <-> COM TxPDO-Map Inputs/Data In 17
//     ComTask Inputs/GVL_COM.K4S6_01_E5_stComIn/D[18] <-> COM TxPDO-Map Inputs/Data In 18
//     ComTask Inputs/GVL_COM.K4S6_01_E5_stComIn/D[19] <-> COM TxPDO-Map Inputs/Data In 19
//     ComTask Inputs/GVL_COM.K4S6_01_E5_stComIn/D[1] <-> COM TxPDO-Map Inputs/Data In 1
//     ComTask Inputs/GVL_COM.K4S6_01_E5_stComIn/D[20] <-> COM TxPDO-Map Inputs/Data In 20
//     ComTask Inputs/GVL_COM.K4S6_01_E5_stComIn/D[21] <-> COM TxPDO-Map Inputs/Data In 21
//     ComTask Inputs/GVL_COM.K4S6_01_E5_stComIn/D[2] <-> COM TxPDO-Map Inputs/Data In 2
//     ComTask Inputs/GVL_COM.K4S6_01_E5_stComIn/D[3] <-> COM TxPDO-Map Inputs/Data In 3
//     ComTask Inputs/GVL_COM.K4S6_01_E5_stComIn/D[4] <-> COM TxPDO-Map Inputs/Data In 4
//     ComTask Inputs/GVL_COM.K4S6_01_E5_stComIn/D[5] <-> COM TxPDO-Map Inputs/Data In 5
//     ComTask Inputs/GVL_COM.K4S6_01_E5_stComIn/D[6] <-> COM TxPDO-Map Inputs/Data In 6
//     ComTask Inputs/GVL_COM.K4S6_01_E5_stComIn/D[7] <-> COM TxPDO-Map Inputs/Data In 7
//     ComTask Inputs/GVL_COM.K4S6_01_E5_stComIn/D[8] <-> COM TxPDO-Map Inputs/Data In 8
//     ComTask Inputs/GVL_COM.K4S6_01_E5_stComIn/D[9] <-> COM TxPDO-Map Inputs/Data In 9
//     ComTask Inputs/GVL_COM.K4S6_01_E5_stComIn/Status <-> COM TxPDO-Map Inputs/Status
//     ComTask Outputs/GVL_COM.K4S6_01_E5_stComOut/Ctrl <-> COM RxPDO-Map Outputs/Ctrl
//     ComTask Outputs/GVL_COM.K4S6_01_E5_stComOut/D[0] <-> COM RxPDO-Map Outputs/Data Out 0
//     ComTask Outputs/GVL_COM.K4S6_01_E5_stComOut/D[10] <-> COM RxPDO-Map Outputs/Data Out 10
//     ComTask Outputs/GVL_COM.K4S6_01_E5_stComOut/D[11] <-> COM RxPDO-Map Outputs/Data Out 11
//     ComTask Outputs/GVL_COM.K4S6_01_E5_stComOut/D[12] <-> COM RxPDO-Map Outputs/Data Out 12
//     ComTask Outputs/GVL_COM.K4S6_01_E5_stComOut/D[13] <-> COM RxPDO-Map Outputs/Data Out 13
//     ComTask Outputs/GVL_COM.K4S6_01_E5_stComOut/D[14] <-> COM RxPDO-Map Outputs/Data Out 14
//     ComTask Outputs/GVL_COM.K4S6_01_E5_stComOut/D[15] <-> COM RxPDO-Map Outputs/Data Out 15
//     ComTask Outputs/GVL_COM.K4S6_01_E5_stComOut/D[16] <-> COM RxPDO-Map Outputs/Data Out 16
//     ComTask Outputs/GVL_COM.K4S6_01_E5_stComOut/D[17] <-> COM RxPDO-Map Outputs/Data Out 17
//     ComTask Outputs/GVL_COM.K4S6_01_E5_stComOut/D[18] <-> COM RxPDO-Map Outputs/Data Out 18
//     ComTask Outputs/GVL_COM.K4S6_01_E5_stComOut/D[19] <-> COM RxPDO-Map Outputs/Data Out 19
//     ComTask Outputs/GVL_COM.K4S6_01_E5_stComOut/D[1] <-> COM RxPDO-Map Outputs/Data Out 1
//     ComTask Outputs/GVL_COM.K4S6_01_E5_stComOut/D[20] <-> COM RxPDO-Map Outputs/Data Out 20
//     ComTask Outputs/GVL_COM.K4S6_01_E5_stComOut/D[21] <-> COM RxPDO-Map Outputs/Data Out 21
//     ComTask Outputs/GVL_COM.K4S6_01_E5_stComOut/D[2] <-> COM RxPDO-Map Outputs/Data Out 2
//     ComTask Outputs/GVL_COM.K4S6_01_E5_stComOut/D[3] <-> COM RxPDO-Map Outputs/Data Out 3
//     ComTask Outputs/GVL_COM.K4S6_01_E5_stComOut/D[4] <-> COM RxPDO-Map Outputs/Data Out 4
//     ComTask Outputs/GVL_COM.K4S6_01_E5_stComOut/D[5] <-> COM RxPDO-Map Outputs/Data Out 5
//     ComTask Outputs/GVL_COM.K4S6_01_E5_stComOut/D[6] <-> COM RxPDO-Map Outputs/Data Out 6
//     ComTask Outputs/GVL_COM.K4S6_01_E5_stComOut/D[7] <-> COM RxPDO-Map Outputs/Data Out 7
//     ComTask Outputs/GVL_COM.K4S6_01_E5_stComOut/D[8] <-> COM RxPDO-Map Outputs/Data Out 8
//     ComTask Outputs/GVL_COM.K4S6_01_E5_stComOut/D[9] <-> COM RxPDO-Map Outputs/Data Out 9
//   plc_tmo_hutch_vac Instance <-> Device 1 (EtherCAT)/TMO_K4S6_DRL_01 (EK1100)/K4S6_01_E6 (EL1004)
//     PlcTask Inputs/GVL_Hutch_Pumps.LI3K4_IP1_OUT_PTM_01.i_xAtSpd <-> Channel 1/Input
//     PlcTask Inputs/GVL_Hutch_Pumps.LI3K4_IP1_OUT_PTM_01.i_xFaultNC <-> Channel 3/Input
//     PlcTask Inputs/GVL_Hutch_Pumps.LI3K4_IP1_OUT_PTM_01.i_xRemote <-> Channel 2/Input
//     PlcTask Inputs/GVL_Hutch_Pumps.TM1K4_PTM_01.i_xAtSpd <-> Channel 4/Input
//   plc_tmo_hutch_vac Instance <-> Device 1 (EtherCAT)/TMO_K4S6_DRL_01 (EK1100)/K4S6_01_E7 (EL2004)
//     PlcTask Outputs/GVL_Hutch_Pumps.LI3K4_IP1_OUT_PTM_01.q_PumpingStation <-> Channel 3/Output
//     PlcTask Outputs/GVL_Hutch_Pumps.LI3K4_IP1_OUT_PTM_01.q_RunDO <-> Channel 1/Output
//     PlcTask Outputs/GVL_Hutch_Pumps.LI3K4_IP1_OUT_PTM_01.q_xRemote <-> Channel 2/Output
//     PlcTask Outputs/GVL_Hutch_Pumps.TM1K4_PTM_01.q_RunDO <-> Channel 4/Output
//   plc_tmo_hutch_vac Instance <-> Device 1 (EtherCAT)/TMO_K4S6_DRL_01 (EK1100)/K4S6_01_E8 (EL1004)
//     PlcTask Inputs/GVL_Hutch_Pumps.IM5K4_PPM_PTM_01.i_xAtSpd <-> Channel 3/Input
//     PlcTask Inputs/GVL_Hutch_Pumps.IM5K4_PPM_PTM_01.i_xRemote <-> Channel 4/Input
//     PlcTask Inputs/GVL_Hutch_Pumps.TM1K4_PTM_01.i_xFaultNC <-> Channel 2/Input
//     PlcTask Inputs/GVL_Hutch_Pumps.TM1K4_PTM_01.i_xRemote <-> Channel 1/Input
//   plc_tmo_hutch_vac Instance <-> Device 1 (EtherCAT)/TMO_K4S6_DRL_01 (EK1100)/K4S6_01_E9 (EL2004)
//     PlcTask Outputs/GVL_Hutch_Pumps.IM5K4_PPM_PTM_01.q_RunDO <-> Channel 3/Output
//     PlcTask Outputs/GVL_Hutch_Pumps.IM5K4_PPM_PTM_01.q_xRemote <-> Channel 4/Output
//     PlcTask Outputs/GVL_Hutch_Pumps.TM1K4_PTM_01.q_PumpingStation <-> Channel 2/Output
//     PlcTask Outputs/GVL_Hutch_Pumps.TM1K4_PTM_01.q_xRemote <-> Channel 1/Output
//   plc_tmo_hutch_vac Instance <-> Device 1 (EtherCAT)/TMO_K4S8_DRL_01 (EK1100)/K4S8_01_E1 (EL1004)
//     FSVTask Inputs/GVL_FS_Devices.MR4K4_KBO_VFS_1.i_xClsLS <-> Channel 1/Input
//     FSVTask Inputs/GVL_FS_Devices.MR4K4_KBO_VFS_1.i_xOpnLS <-> Channel 2/Input
//   plc_tmo_hutch_vac Instance <-> Device 1 (EtherCAT)/TMO_K4S8_DRL_01 (EK1100)/K4S8_01_E3 (EL2202)
//     FSVTask Outputs/GVL_FS_Devices.MR4K4_KBO_VFS_1.q_xClose_A <-> Channel 1/Output
//     FSVTask Outputs/GVL_FS_Devices.MR4K4_KBO_VFS_1.q_xClose_B <-> Channel 2/Output
//   plc_tmo_hutch_vac Instance <-> Device 1 (EtherCAT)/TMO_K4S8_DRL_01 (EK1100)/K4S8_01_E4 (EL2202)
//     FSVTask Outputs/GVL_FS_Devices.MR4K4_KBO_VFS_1.q_xClose_C <-> Channel 1/Output
//     FSVTask Outputs/GVL_FS_Devices.MR4K4_KBO_VFS_1.q_xOPN_DO <-> Channel 2/Output
//   plc_tmo_hutch_vac Instance <-> Device 1 (EtherCAT)/TMO_K4S8_DRL_01 (EK1100)/K4S8_01_E5 (EL1004)
//     ComTask Inputs/GVL_Hutch_Valves.MR4K4_KBO_VWC_01.i_xClsLS <-> Channel 2/Input
//     ComTask Inputs/GVL_Hutch_Valves.MR5K4_KBO_VWC_01.i_xClsLS <-> Channel 4/Input
//     ComTask Inputs/GVL_Hutch_Valves.MR4K4_KBO_VWC_01.i_xOpnLS <-> Channel 1/Input
//     ComTask Inputs/GVL_Hutch_Valves.MR5K4_KBO_VWC_01.i_xOpnLS <-> Channel 3/Input
//   plc_tmo_hutch_vac Instance <-> Device 1 (EtherCAT)/TMO_K4S8_DRL_01 (EK1100)/K4S8_01_E6 (EL2004)
//     ComTask Outputs/GVL_Hutch_Valves.MR4K4_KBO_VWC_01.q_xOPN_DO <-> Channel 1/Output
//     ComTask Outputs/GVL_Hutch_Valves.MR5K4_KBO_VWC_01.q_xOPN_DO <-> Channel 2/Output
//   plc_tmo_hutch_vac Instance <-> Device 1 (EtherCAT)/TMO_WALL_WEST_EP01 (EP4374-0002)
//     ComTask Outputs/GVL_Hutch_Valves.TMO_ROUGH1_VFV_01.q_iRawPosition <-> AO Outputs Channel 3/Analog output
//     PlcTask Inputs/GVL_Hutch_Gauges.TMO_ROUGH1_GPI_01.i_iPRESS_R <-> AI Inputs Channel 1/Value
//     PlcTask Inputs/GVL_Hutch_Gauges.TMO_ROUGH2_GPI_01.i_iPRESS_R <-> AI Inputs Channel 2/Value

CONFIGURATION plc_tmo_hutch_vac
    RESOURCE PLC ON TwinCAT3
        TASK ComTask(INTERVAL := T#3ms, PRIORITY := 21);
        TASK FSVTask(INTERVAL := T#1ms, PRIORITY := 1);
        TASK PlcTask(INTERVAL := T#10ms, PRIORITY := 20);
        PROGRAM PRG_COM WITH ComTask : PRG_COM;
        PROGRAM PRG_FSV WITH FSVTask : PRG_FSV;
        PROGRAM MAIN WITH PlcTask : MAIN;
    END_RESOURCE
END_CONFIGURATION

// ---- GVLs/GVL_Hutch_Gauges.TcGVL
//{attribute 'qualified_only'}
VAR_GLOBAL
(* Pirani & Cold Cathode*)

	{attribute 'pytmc' :=' pv: MR2K4:KBO:GPI:01 '}
	{attribute 'TcLinkTo' := 	'.i_iPRESS_R	:=	TIIB[TMO_K4S2_DRL_02 (EK1100)]^K4S2_02_E1 (EL3174)^AI Standard Channel 2^Value '}
	MR2K4_KBO_GPI_01 : FB_MKS275;
	
	{attribute 'pytmc' :=' pv: TV1K4:GCC:01 '}
	{attribute 'TcLinkTo' := 	'.i_iPRESS_R	:=	TIIB[TMO_K4S2_DRL_02 (EK1100)]^K4S2_02_E1 (EL3174)^AI Standard Channel 3^Value;
								 .i_xHV_ON	    :=	TIIB[TMO_K4S2_DRL_02 (EK1100)]^K4S2_02_E7 (EL1124)^Channel 3^Input;
								 .i_xDisc_Active:=	TIIB[TMO_K4S2_DRL_02 (EK1100)]^K4S2_02_E7 (EL1124)^Channel 4^Input;								 
								 .q_xHV_DIS		:= 	TIIB[TMO_K4S2_DRL_02 (EK1100)]^K4S2_02_E5 (EL2624)^Channel 2^Output	'}	
	MR2K4_KBO_GCC_01 : FB_MKS500;
	
	{attribute 'pytmc' :=' pv: PA1K4:IP1:GPI:01 '}
	{attribute 'TcLinkTo' := 	'.i_iPRESS_R	:=	TIIB[TMO_K4S2_DRL_02 (EK1100)]^K4S2_02_E2 (EL3174)^AI Standard Channel 1^Value '}	
	PA1K4_IP1_GPI_01 : FB_MKS275;
	

	{attribute 'pytmc' :=' pv: PA1K4:IP1:GCC:01 '}
	{attribute 'TcLinkTo' := 	'.i_iPRESS_R	:=	TIIB[TMO_K4S2_DRL_02 (EK1100)]^K4S2_02_E1 (EL3174)^AI Standard Channel 4^Value;
								 .i_xHV_ON	    :=	TIIB[TMO_K4S2_DRL_02 (EK1100)]^K4S2_02_E8 (EL1124)^Channel 1^Input;
								 .i_xDisc_Active:=	TIIB[TMO_K4S2_DRL_02 (EK1100)]^K4S2_02_E8 (EL1124)^Channel 2^Input;								 
								 .q_xHV_DIS		:= 	TIIB[TMO_K4S2_DRL_02 (EK1100)]^K4S2_02_E5 (EL2624)^Channel 3^Output	'}		
	PA1K4_IP1_GCC_01 : FB_MKS500;
	

	{attribute 'pytmc' :=' pv: IM4K4:PPM:GCC:01 '}
	{attribute 'TcLinkTo' := 	'.i_iPRESS_R	:=	TIIB[TMO_K4S2_DRL_02 (EK1100)]^K4S2_02_E2 (EL3174)^AI Standard Channel 2^Value;
								 .i_xHV_ON	    :=	TIIB[TMO_K4S2_DRL_02 (EK1100)]^K4S2_02_E8 (EL1124)^Channel 3^Input;
								 .i_xDisc_Active:=	TIIB[TMO_K4S2_DRL_02 (EK1100)]^K4S2_02_E8 (EL1124)^Channel 4^Input;								 
								 .q_xHV_DIS		:= 	TIIB[TMO_K4S2_DRL_02 (EK1100)]^K4S2_02_E5 (EL2624)^Channel 4^Output	'}			
	IM4K4_PPM_GCC_01 : FB_MKS500;
	

    LI2K4_IP1_GFS_01 : FB_MKS422;
	
	
	{attribute 'pytmc' :=' pv: TM4K4:GCC:01 '}
	{attribute 'TcLinkTo' := 	'.i_iPRESS_R	:=	TIIB[TMO_K4S6_DRL_01 (EK1100)]^K4S6_01_E15 (EL3174)^AI Standard Channel 1^Value;
								 .i_xHV_ON	    :=	TIIB[TMO_K4S6_DRL_01 (EK1100)]^K4S6_01_E20 (EL1124)^Channel 1^Input;
								 .i_xDisc_Active:=	TIIB[TMO_K4S6_DRL_01 (EK1100)]^K4S6_01_E20 (EL1124)^Channel 2^Input;								 
								 .q_xHV_DIS		:= 	TIIB[TMO_K4S6_DRL_01 (EK1100)]^K4S6_01_E14 (EL2624)^Channel 1^Output	'}		
	TM1K4_GCC_01 : FB_MKS500;
	
	{attribute 'pytmc' :=' pv: IM5K4:PPM:GCC:01 '}
	{attribute 'TcLinkTo' := 	'.i_iPRESS_R	:=	TIIB[TMO_K4S6_DRL_01 (EK1100)]^K4S6_01_E15 (EL3174)^AI Standard Channel 2^Value;
								 .i_xHV_ON	    :=	TIIB[TMO_K4S6_DRL_01 (EK1100)]^K4S6_01_E20 (EL1124)^Channel 3^Input;
								 .i_xDisc_Active:=	TIIB[TMO_K4S6_DRL_01 (EK1100)]^K4S6_01_E20 (EL1124)^Channel 4^Input;								 
								 .q_xHV_DIS		:= 	TIIB[TMO_K4S6_DRL_01 (EK1100)]^K4S6_01_E14 (EL2624)^Channel 2^Output	'}		
	IM5K4_PPM_GCC_01 : FB_MKS500;
	
	
	{attribute 'pytmc' :=' pv: PA2K4:IP1:GPI:01 '}
	{attribute 'TcLinkTo' := 	'.i_iPRESS_R	:=	TIIB[TMO_K4S6_DRL_01 (EK1100)]^K4S6_01_E15 (EL3174)^AI Standard Channel 4^Value '}	
	PA2K4_IP1_GPI_01 : FB_MKS275;
	
	{attribute 'pytmc' :=' pv: PA2K4:IP1:GCC:01 '}
	{attribute 'TcLinkTo' := 	'.i_iPRESS_R	:=	TIIB[TMO_K4S6_DRL_01 (EK1100)]^K4S6_01_E15 (EL3174)^AI Standard Channel 3^Value;
								 .i_xHV_ON	    :=	TIIB[TMO_K4S6_DRL_01 (EK1100)]^K4S6_01_E21 (EL1124)^Channel 1^Input;
								 .i_xDisc_Active:=	TIIB[TMO_K4S6_DRL_01 (EK1100)]^K4S6_01_E21 (EL1124)^Channel 2^Input;								 
								 .q_xHV_DIS		:= 	TIIB[TMO_K4S6_DRL_01 (EK1100)]^K4S6_01_E14 (EL2624)^Channel 3^Output	'}		
	PA2K4_IP1_GCC_01 : FB_MKS500;


	{attribute 'pytmc' :=' pv: MR4K4:KBO:GPI:01 '}
	{attribute 'TcLinkTo' := 	'.i_iPRESS_R	:=	TIIB[TMO_K4S6_DRL_01 (EK1100)]^K4S6_01_E18 (EL3174)^AI Standard Channel 1^Value '}		
	MR4K4_KBO_GPI_01 : FB_MKS275;

	{attribute 'pytmc' :=' pv: MR4K4:KBO:GCC:01 '}
	{attribute 'TcLinkTo' := 	'.i_iPRESS_R	:=	TIIB[TMO_K4S6_DRL_01 (EK1100)]^K4S6_01_E18 (EL3174)^AI Standard Channel 2^Value;
								 .i_xHV_ON	    :=	TIIB[TMO_K4S6_DRL_01 (EK1100)]^K4S6_01_E21 (EL1124)^Channel 3^Input;
								 .i_xDisc_Active:=	TIIB[TMO_K4S6_DRL_01 (EK1100)]^K4S6_01_E21 (EL1124)^Channel 4^Input;								 
								 .q_xHV_DIS		:= 	TIIB[TMO_K4S6_DRL_01 (EK1100)]^K4S6_01_E14 (EL2624)^Channel 4^Output	'}			
	MR4K4_KBO_GCC_01 : FB_MKS500;
	
	(* Roughing gauges *)

	{attribute 'pytmc' :=' pv: TMO:ROUGH1:GPI:01 '}
	{attribute 'TcLinkTo' := 	'.i_iPRESS_R	:=	TIIB[TMO_WALL_WEST_EP01 (EP4374-0002)]^AI Inputs Channel 1^Value	'}	
	TMO_ROUGH1_GPI_01 : FB_9XX;
	
	{attribute 'pytmc' :=' pv: TMO:ROUGH1:GPI:02 '}
	{attribute 'TcLinkTo' := 	'.i_iPRESS_R	:=	TIIB[TMO_K4S2_ EP1 (EP4374-0002)]^AI Inputs Channel 1^Value	'}	
	TMO_ROUGH1_GPI_02 : FB_9XX;
	
	{attribute 'pytmc' :=' pv: TMO:ROUGH1:GPI:03 '}
	{attribute 'TcLinkTo' := 	'.i_iPRESS_R	:=	TIIB[TMO_K4S6_ EP1 (EP4374-0002)]^AI Inputs Channel 1^Value	'}		
	TMO_ROUGH1_GPI_03 : FB_9XX;

	{attribute 'pytmc' :=' pv: TMO:ROUGH2:GPI:01 '}
	{attribute 'TcLinkTo' := 	'.i_iPRESS_R	:=	TIIB[TMO_WALL_WEST_EP01 (EP4374-0002)]^AI Inputs Channel 2^Value	'}	
	TMO_ROUGH2_GPI_01 : FB_9XX;
	
	{attribute 'pytmc' :=' pv: TMO:ROUGH2:GPI:02 '}
	{attribute 'TcLinkTo' := 	'.i_iPRESS_R	:=	TIIB[TMO_K4S2_ EP1 (EP4374-0002)]^AI Inputs Channel 2^Value	'}	
	TMO_ROUGH2_GPI_02 : FB_9XX;	
	
	
	

END_VAR

// ---- GVLs/GVL_Hutch_Pumps.TcGVL
//{attribute 'qualified_only'}
VAR_GLOBAL
	
	
(* Ion pumps *)

	MR2K4_KBO_PIP_01 : FB_PIP_Gamma;
	
	MR4K4_KBO_PIP_01 : FB_PIP_Gamma;
	
	PA2K4_IP1_PIP_01 : FB_PIP_Gamma;
	

(* Granite 1 *)
(* Pfeiffer Turbo Pumps TC110 *)

	{attribute 'TcLinkTo' := 	'.i_xAtSpd			:=	TIIB[TMO_K4S2_DRL_02 (EK1100)]^K4S2_02_E11 (EL1004)^Channel 2^Input;
								 .i_xFaultNC		:=	TIIB[TMO_K4S2_DRL_02 (EK1100)]^K4S2_02_E11 (EL1004)^Channel 1^Input;
								 .q_RunDO			:=	TIIB[TMO_K4S2_DRL_02 (EK1100)]^K4S2_02_E12 (EL2794)^Channel 1^Output;
								 .q_xReset 			:=	TIIB[TMO_K4S2_DRL_02 (EK1100)]^K4S2_02_E12 (EL2794)^Channel 2^Output				 
	'}
	{attribute 'pytmc' := '
		pv: PA1K4:IP1:PTM:01
		io: io
	'}
	PA1K4_IP1_PTM_01 : FB_PTM_Pfeiffer;



	{attribute 'TcLinkTo' := 	'.i_xAtSpd			:=	TIIB[TMO_K4S2_DRL_02 (EK1100)]^K4S2_02_E11 (EL1004)^Channel 4^Input;
								 .i_xFaultNC		:=	TIIB[TMO_K4S2_DRL_02 (EK1100)]^K4S2_02_E11 (EL1004)^Channel 3^Input;
								 .q_RunDO			:=	TIIB[TMO_K4S2_DRL_02 (EK1100)]^K4S2_02_E12 (EL2794)^Channel 3^Output;
								 .q_xReset 			:=	TIIB[TMO_K4S2_DRL_02 (EK1100)]^K4S2_02_E12 (EL2794)^Channel 4^Output				 
	'}
	{attribute 'pytmc' := '
		pv: PA1K4:IP1:PTM:02
		io: io
	'}	
	PA1K4_IP1_PTM_02 : FB_PTM_Pfeiffer;
	
	{attribute 'TcLinkTo' := 	'.i_xAtSpd			:=	TIIB[TMO_K4S2_DRL_02 (EK1100)]^K4S2_02_E13 (EL1004)^Channel 2^Input;
								 .i_xFaultNC		:=	TIIB[TMO_K4S2_DRL_02 (EK1100)]^K4S2_02_E13 (EL1004)^Channel 1^Input;
								 .q_RunDO			:=	TIIB[TMO_K4S2_DRL_02 (EK1100)]^K4S2_02_E14 (EL2794)^Channel 1^Output;
								 .q_xReset 			:=	TIIB[TMO_K4S2_DRL_02 (EK1100)]^K4S2_02_E14 (EL2794)^Channel 2^Output				 
	'}
	{attribute 'pytmc' := '
		pv: PA1K4:IP1:PTM:03
		io: io
	'}	
	PA1K4_IP1_PTM_03 : FB_PTM_Pfeiffer;
	
	// They share the same serial port
	st_Pfeiffer_CTRL_PTM_01_02_03			: ARRAY[1..20] OF ST_PfeifferControl;
	st_Pfeiffer_RBK_PTM_01_02_03			: ARRAY[1..20] OF ST_PfeifferStatus;
	PA1K4_IP1_PTM_01_02_03_COM: FB_PFEIFFER_COM;

(* Leybold Turbo Pumps Mag.drive is*)	

	{attribute 'TcLinkTo' := 	'.i_xAtSpd			:=	TIIB[TMO_K4S2_DRL_02 (EK1100)]^K4S2_02_E15 (EL1004)^Channel 2^Input;
								 .i_xFaultNC		:=	TIIB[TMO_K4S2_DRL_02 (EK1100)]^K4S2_02_E15 (EL1004)^Channel 1^Input;
								 .q_RunDO			:=	TIIB[TMO_K4S2_DRL_02 (EK1100)]^K4S2_02_E16 (EL2794)^Channel 1^Output			 
	'}
	{attribute 'pytmc' := '
		pv: IM4K4:PPM:PTM:01
		io: io
	'}
	IM4K4_PPM_PTM_01 : FB_PTM_TurboDrive;
	IM4K4_PPM_PTM_01_COM:FB_Oerlikon_TD20_COM;
	
	{attribute 'TcLinkTo' := 	'.i_xAtSpd			:=	TIIB[TMO_K4S2_DRL_02 (EK1100)]^K4S2_02_E15 (EL1004)^Channel 4^Input;
								 .i_xFaultNC		:=	TIIB[TMO_K4S2_DRL_02 (EK1100)]^K4S2_02_E15 (EL1004)^Channel 3^Input;
								 .q_RunDO			:=	TIIB[TMO_K4S2_DRL_02 (EK1100)]^K4S2_02_E16 (EL2794)^Channel 2^Output			 
	'}
	{attribute 'pytmc' := '
		pv: LI1K4:IP1:PTM:01
		io: io
	'}
	LI1K4_IP1_PTM_01 : FB_PTM_TurboDrive;
	LI1K4_IP1_PTM_01_COM: FB_Oerlikon_TD20_COM;

(* Granite 2 *)
(* Pfeiffer Turbo Pumps TM700 *)

	{attribute 'TcLinkTo' := 	'.i_xAtSpd			:=	TIIB[TMO_K4S6_DRL_01 (EK1100)]^K4S6_01_E6 (EL1004)^Channel 1^Input;
								 .i_xRemote			:=	TIIB[TMO_K4S6_DRL_01 (EK1100)]^K4S6_01_E6 (EL1004)^Channel 2^Input;
								 .i_xFaultNC		:=	TIIB[TMO_K4S6_DRL_01 (EK1100)]^K4S6_01_E6 (EL1004)^Channel 3^Input;
								 .q_RunDO			:=	TIIB[TMO_K4S6_DRL_01 (EK1100)]^K4S6_01_E7 (EL2004)^Channel 1^Output;
								 .q_xRemote			:=	TIIB[TMO_K4S6_DRL_01 (EK1100)]^K4S6_01_E7 (EL2004)^Channel 2^Output;
								 .q_PumpingStation	:=	TIIB[TMO_K4S6_DRL_01 (EK1100)]^K4S6_01_E7 (EL2004)^Channel 3^Output				 
	'}
	{attribute 'pytmc' := '
		pv: LI3K4:IP1:OUT:PTM:01
		io: io
	'}
    LI3K4_IP1_OUT_PTM_01 : FB_PTM_Pfeiffer;
(* Pfeiffer Turbo Pumps TC400 *)
	
	{attribute 'TcLinkTo' := 	'.i_xAtSpd			:=	TIIB[TMO_K4S6_DRL_01 (EK1100)]^K4S6_01_E6 (EL1004)^Channel 4^Input;
								 .i_xRemote			:=	TIIB[TMO_K4S6_DRL_01 (EK1100)]^K4S6_01_E8 (EL1004)^Channel 1^Input;
								 .i_xFaultNC		:=	TIIB[TMO_K4S6_DRL_01 (EK1100)]^K4S6_01_E8 (EL1004)^Channel 2^Input;					 
								 .q_RunDO			:=	TIIB[TMO_K4S6_DRL_01 (EK1100)]^K4S6_01_E7 (EL2004)^Channel 4^Output;
								 .q_xRemote			:=	TIIB[TMO_K4S6_DRL_01 (EK1100)]^K4S6_01_E9 (EL2004)^Channel 1^Output;
								 .q_PumpingStation	:=	TIIB[TMO_K4S6_DRL_01 (EK1100)]^K4S6_01_E9 (EL2004)^Channel 2^Output				 
	'}
	{attribute 'pytmc' := '
		pv: TM1K4:PTM:01
		io: io
	'}
	TM1K4_PTM_01 : FB_PTM_Pfeiffer;
	
	
	{attribute 'TcLinkTo' := 	'.i_xAtSpd			:=	TIIB[TMO_K4S6_DRL_01 (EK1100)]^K4S6_01_E8 (EL1004)^Channel 3^Input;
								 .i_xRemote			:=	TIIB[TMO_K4S6_DRL_01 (EK1100)]^K4S6_01_E8 (EL1004)^Channel 4^Input;
								 .i_xFaultNC		:=	TIIB[TMO_K4S6_DRL_01 (EK1100)]^K4S6_01_E11 (EL1004)^Channel 1^Input;
								 .q_RunDO			:=	TIIB[TMO_K4S6_DRL_01 (EK1100)]^K4S6_01_E9 (EL2004)^Channel 3^Output;
								 .q_xRemote			:=	TIIB[TMO_K4S6_DRL_01 (EK1100)]^K4S6_01_E9 (EL2004)^Channel 4^Output;
								 .q_PumpingStation	:=	TIIB[TMO_K4S6_DRL_01 (EK1100)]^K4S6_01_E12 (EL2004)^Channel 1^Output				 
	'}
	{attribute 'pytmc' := '
		pv: IM5K4:PPM:PTM:01
		io: io
	'}
	IM5K4_PPM_PTM_01 : FB_PTM_Pfeiffer;
	// They share the same serial port
	st_Pfeiffer_CTRL_PTM_Granite2			: ARRAY[1..20] OF ST_PfeifferControl;
	st_Pfeiffer_RBK_PTM_Granite2			: ARRAY[1..20] OF ST_PfeifferStatus;
	Granite2_PTM_COM :FB_PFEIFFER_COM;
	
END_VAR

// ---- GVLs/GVL_Hutch_Valves.TcGVL
//{attribute 'qualified_only'}
VAR_GLOBAL
	
(*  Beamline Windows Valve *)

	{attribute 'pytmc' :=' pv: MR2K4:KBO:VWC:01 '}
	{attribute 'TcLinkTo' := 	'.i_xOpnLS	:=	TIIB[TMO_K4S2_DRL_01 (EK1100)]^K4S2_01_E5 (EL1004)^Channel 1^Input;
								 .i_xClsLS	:=	TIIB[TMO_K4S2_DRL_01 (EK1100)]^K4S2_01_E5 (EL1004)^Channel 2^Input;
								.q_xOPN_DO	:=	TIIB[TMO_K4S2_DRL_01 (EK1100)]^K4S2_01_E6 (EL2004)^Channel 1^Output'}
	MR2K4_KBO_VWC_01 : FB_VGC_2S;
	
	
	{attribute 'pytmc' :=' pv: MR3K4:KBO:VWC:01 '}
	{attribute 'TcLinkTo' := 	'.i_xOpnLS	:=	TIIB[TMO_K4S2_DRL_01 (EK1100)]^K4S2_01_E5 (EL1004)^Channel 3^Input;
								 .i_xClsLS	:=	TIIB[TMO_K4S2_DRL_01 (EK1100)]^K4S2_01_E5 (EL1004)^Channel 4^Input;
								.q_xOPN_DO	:=	TIIB[TMO_K4S2_DRL_01 (EK1100)]^K4S2_01_E6 (EL2004)^Channel 2^Output'}	
	MR3K4_KBO_VWC_01 : FB_VGC_2S;
	
	
	{attribute 'pytmc' :=' pv: LI3K4:IP1:VWC:01 '}
	{attribute 'TcLinkTo' := 	'.i_xOpnLS	:=	TIIB[TMO_K4S6_DRL_01 (EK1100)]^K4S6_01_E3 (EL1004)^Channel 1^Input;
								 .i_xClsLS	:=	TIIB[TMO_K4S6_DRL_01 (EK1100)]^K4S6_01_E3 (EL1004)^Channel 2^Input;
								.q_xOPN_DO	:=	TIIB[TMO_K4S6_DRL_01 (EK1100)]^K4S6_01_E4 (EL2004)^Channel 1^Output'}		
	LI3K4_IP1_VWC_01 : FB_VGC_2S;
	
	{attribute 'pytmc' :=' pv: PC5K4:VWC:01 '}
	{attribute 'TcLinkTo' := 	'.i_xOpnLS	:=	TIIB[TMO_K4S6_DRL_01 (EK1100)]^K4S6_01_E3 (EL1004)^Channel 3^Input;
								 .i_xClsLS	:=	TIIB[TMO_K4S6_DRL_01 (EK1100)]^K4S6_01_E3 (EL1004)^Channel 4^Input;
								.q_xOPN_DO	:=	TIIB[TMO_K4S6_DRL_01 (EK1100)]^K4S6_01_E4 (EL2004)^Channel 2^Output'}		
	PC5K4_VWC_01 : FB_VGC_2S;


	{attribute 'pytmc' :=' pv: MR4K4:KBO:VWC:01 '}
	{attribute 'TcLinkTo' := 	'.i_xOpnLS	:=	TIIB[TMO_K4S8_DRL_01 (EK1100)]^K4S8_01_E5 (EL1004)^Channel 1^Input;
								 .i_xClsLS	:=	TIIB[TMO_K4S8_DRL_01 (EK1100)]^K4S8_01_E5 (EL1004)^Channel 2^Input;
								.q_xOPN_DO	:=	TIIB[TMO_K4S8_DRL_01 (EK1100)]^K4S8_01_E6 (EL2004)^Channel 1^Output'}		
	MR4K4_KBO_VWC_01 : FB_VGC_2S;
	
	
	{attribute 'pytmc' :=' pv: MR5K4:KBO:VWC:01 '}
	{attribute 'TcLinkTo' := 	'.i_xOpnLS	:=	TIIB[TMO_K4S8_DRL_01 (EK1100)]^K4S8_01_E5 (EL1004)^Channel 3^Input;
								 .i_xClsLS	:=	TIIB[TMO_K4S8_DRL_01 (EK1100)]^K4S8_01_E5 (EL1004)^Channel 4^Input;
								.q_xOPN_DO	:=	TIIB[TMO_K4S8_DRL_01 (EK1100)]^K4S8_01_E6 (EL2004)^Channel 2^Output'}		
	MR5K4_KBO_VWC_01 : FB_VGC_2S;
	
(* Not installed yet	
	TM2K4_VWC_01 : FB_VGC;
	
	*)
	
(*  Roughing valve *)	

	{attribute 'pytmc' :=' pv: TMO:ROUGH1:VRC:01 '}
	{attribute 'TcLinkTo' := 	'.i_xOpnLS	:=	TIIB[TMO_K4S2_DRL_02 (EK1100)]^K4S2_02_E19 (EL1004)^Channel 1^Input;
								 .i_xClsLS	:=	TIIB[TMO_K4S2_DRL_02 (EK1100)]^K4S2_02_E19 (EL1004)^Channel 2^Input;
								.q_xOPN_DO	:=	TIIB[TMO_K4S2_DRL_02 (EK1100)]^K4S2_02_E20 (EL2004)^Channel 1^Output'}
	TMO_ROUGH1_VRC_01 : FB_VRC;

	{attribute 'pytmc' :=' pv: TMO:ROUGH1:VRC:02 '}
	{attribute 'TcLinkTo' := 	'.i_xOpnLS	:=	TIIB[TMO_K4S6_DRL_01 (EK1100)]^K4S6_01_E1 (EL1004)^Channel 1^Input;
								 .i_xClsLS	:=	TIIB[TMO_K4S6_DRL_01 (EK1100)]^K4S6_01_E1 (EL1004)^Channel 2^Input;
								.q_xOPN_DO	:=	TIIB[TMO_K4S6_DRL_01 (EK1100)]^K4S6_01_E2 (EL2004)^Channel 1^Output'}
	TMO_ROUGH1_VRC_02 : FB_VRC;
	
	{attribute 'pytmc' :=' pv: TMO:ROUGH2:VRC:01 '}
	{attribute 'TcLinkTo' := 	'.i_xOpnLS	:=	TIIB[TMO_K4S2_DRL_02 (EK1100)]^K4S2_02_E19 (EL1004)^Channel 3^Input;
								 .i_xClsLS	:=	TIIB[TMO_K4S2_DRL_02 (EK1100)]^K4S2_02_E19 (EL1004)^Channel 4^Input;
								.q_xOPN_DO	:=	TIIB[TMO_K4S2_DRL_02 (EK1100)]^K4S2_02_E20 (EL2004)^Channel 2^Output'}
	TMO_ROUGH2_VRC_01 : FB_VRC;

(* MKS248 with MKS1249 solenoid driver *)

	{attribute 'pytmc' :=' pv: TMO:ROUGH1:VFV:01 '}
	{attribute 'TcLinkTo' := 	'.q_iRawPosition	:=	TIIB[TMO_WALL_WEST_EP01 (EP4374-0002)]^AO Outputs Channel 3^Analog output	'}	
     TMO_ROUGH1_VFV_01 : FB_MKS248;
	 
	{attribute 'pytmc' :=' pv: TMO:ROUGH1:VFV:02 '}
	{attribute 'TcLinkTo' := 	'.q_iRawPosition	:=	TIIB[TMO_K4S2_ EP1 (EP4374-0002)]^AO Outputs Channel 3^Analog output	'}	
	 TMO_ROUGH1_VFV_02 : FB_MKS248;
	 
	{attribute 'pytmc' :=' pv: TMO:ROUGH1:VFV:03 '}
	{attribute 'TcLinkTo' := 	'.q_iRawPosition	:=	TIIB[TMO_K4S6_ EP1 (EP4374-0002)]^AO Outputs Channel 3^Analog output	'}		 
	 TMO_ROUGH1_VFV_03 : FB_MKS248;
	 
	{attribute 'pytmc' :=' pv: TMO:ROUGH2:VFV:01 '}
	{attribute 'TcLinkTo' := 	'.q_iRawPosition	:=	TIIB[TMO_K4S2_ EP1 (EP4374-0002)]^AO Outputs Channel 4^Analog output	'}		 
	 TMO_ROUGH2_VFV_01 : FB_MKS248;
	 
(* VFS valves *)

	{attribute 'TcLinkTo' :='.q_xPress_OK		:= 	TIPC^plc_tmo_hutch_vac_fs^plc_tmo_hutch_vac_fs Instance^PlcTask Inputs^GVL_FS_Devices.MR3K4_KBO_VFS_1.i_xPress_OK;
							 .q_xOPN_SW			:=  TIPC^plc_tmo_hutch_vac_fs^plc_tmo_hutch_vac_fs Instance^PlcTask Inputs^GVL_FS_Devices.MR3K4_KBO_VFS_1.i_xOPN_SW;
							 .q_xCLS_SW			:=  TIPC^plc_tmo_hutch_vac_fs^plc_tmo_hutch_vac_fs Instance^PlcTask Inputs^GVL_FS_Devices.MR3K4_KBO_VFS_1.i_xCLS_SW;
							 .q_xVAC_FAULT_Reset:= 	TIPC^plc_tmo_hutch_vac_fs^plc_tmo_hutch_vac_fs Instance^PlcTask Inputs^GVL_FS_Devices.MR3K4_KBO_VFS_1.i_xVAC_FAULT_Reset;
							 .q_xOverrideMode	:= 	TIPC^plc_tmo_hutch_vac_fs^plc_tmo_hutch_vac_fs Instance^PlcTask Inputs^GVL_FS_Devices.MR3K4_KBO_VFS_1.i_xOverrideMode;
							 .q_xOverrideOpen	:= 	TIPC^plc_tmo_hutch_vac_fs^plc_tmo_hutch_vac_fs Instance^PlcTask Inputs^GVL_FS_Devices.MR3K4_KBO_VFS_1.i_xOverrideOpen;
							 .i_xTrigger		:=	TIPC^plc_tmo_hutch_vac_fs^plc_tmo_hutch_vac_fs Instance^PlcTask Outputs^GVL_FS_Devices.MR3K4_KBO_VFS_1.q_xTrigger;
							 .i_xVFS_Open		:=	TIPC^plc_tmo_hutch_vac_fs^plc_tmo_hutch_vac_fs Instance^PlcTask Outputs^GVL_FS_Devices.MR3K4_KBO_VFS_1.q_xVFS_Open;
							 .i_xVFS_Closed		:=	TIPC^plc_tmo_hutch_vac_fs^plc_tmo_hutch_vac_fs Instance^PlcTask Outputs^GVL_FS_Devices.MR3K4_KBO_VFS_1.q_xVFS_Closed;
							 .i_xVAC_FAULT_OK	:=	TIPC^plc_tmo_hutch_vac_fs^plc_tmo_hutch_vac_fs Instance^PlcTask Outputs^GVL_FS_Devices.MR3K4_KBO_VFS_1.q_xVAC_FAULT_OK;
							 .i_xMPS_OK			:=  TIPC^plc_tmo_hutch_vac_fs^plc_tmo_hutch_vac_fs Instance^PlcTask Outputs^GVL_FS_Devices.MR3K4_KBO_VFS_1.q_xMPS_OK;
							 .i_eVFS_State		:=	TIPC^plc_tmo_hutch_vac_fs^plc_tmo_hutch_vac_fs Instance^PlcTask Outputs^GVL_FS_Devices.MR3K4_KBO_VFS_1.q_eVFS_State
	'}
	{attribute 'pytmc' := '
		pv: MR3K4:KBO:VFS:1
		io: io
	'}	
	MR3K4_KBO_VFS_1_Interface : FB_VFS_Interface;
	 
		{attribute 'TcLinkTo' :='.q_xPress_OK		:= 	TIPC^plc_tmo_hutch_vac_fs^plc_tmo_hutch_vac_fs Instance^PlcTask Inputs^GVL_FS_Devices.MR4K4_KBO_VFS_1.i_xPress_OK;
							 .q_xOPN_SW			:=  TIPC^plc_tmo_hutch_vac_fs^plc_tmo_hutch_vac_fs Instance^PlcTask Inputs^GVL_FS_Devices.MR4K4_KBO_VFS_1.i_xOPN_SW;
							 .q_xCLS_SW			:=  TIPC^plc_tmo_hutch_vac_fs^plc_tmo_hutch_vac_fs Instance^PlcTask Inputs^GVL_FS_Devices.MR4K4_KBO_VFS_1.i_xCLS_SW;
							 .q_xVAC_FAULT_Reset:= 	TIPC^plc_tmo_hutch_vac_fs^plc_tmo_hutch_vac_fs Instance^PlcTask Inputs^GVL_FS_Devices.MR4K4_KBO_VFS_1.i_xVAC_FAULT_Reset;
							 .q_xOverrideMode	:= 	TIPC^plc_tmo_hutch_vac_fs^plc_tmo_hutch_vac_fs Instance^PlcTask Inputs^GVL_FS_Devices.MR4K4_KBO_VFS_1.i_xOverrideMode;
							 .q_xOverrideOpen	:= 	TIPC^plc_tmo_hutch_vac_fs^plc_tmo_hutch_vac_fs Instance^PlcTask Inputs^GVL_FS_Devices.MR4K4_KBO_VFS_1.i_xOverrideOpen;
							 .i_xTrigger		:=	TIPC^plc_tmo_hutch_vac_fs^plc_tmo_hutch_vac_fs Instance^PlcTask Outputs^GVL_FS_Devices.MR4K4_KBO_VFS_1.q_xTrigger;
							 .i_xVFS_Open		:=	TIPC^plc_tmo_hutch_vac_fs^plc_tmo_hutch_vac_fs Instance^PlcTask Outputs^GVL_FS_Devices.MR4K4_KBO_VFS_1.q_xVFS_Open;
							 .i_xVFS_Closed		:=	TIPC^plc_tmo_hutch_vac_fs^plc_tmo_hutch_vac_fs Instance^PlcTask Outputs^GVL_FS_Devices.MR4K4_KBO_VFS_1.q_xVFS_Closed;
							 .i_xVAC_FAULT_OK	:=	TIPC^plc_tmo_hutch_vac_fs^plc_tmo_hutch_vac_fs Instance^PlcTask Outputs^GVL_FS_Devices.MR4K4_KBO_VFS_1.q_xVAC_FAULT_OK;
							 .i_xMPS_OK			:=  TIPC^plc_tmo_hutch_vac_fs^plc_tmo_hutch_vac_fs Instance^PlcTask Outputs^GVL_FS_Devices.MR4K4_KBO_VFS_1.q_xMPS_OK;
							 .i_eVFS_State		:=	TIPC^plc_tmo_hutch_vac_fs^plc_tmo_hutch_vac_fs Instance^PlcTask Outputs^GVL_FS_Devices.MR4K4_KBO_VFS_1.q_eVFS_State
	'}
	{attribute 'pytmc' := '
		pv: MR4K4:KBO:VFS:1
		io: io
	'}	
	MR4K4_KBO_VFS_1_Interface : FB_VFS_Interface;
	
	
END_VAR

// ---- GVLs/GVL_Variables.TcGVL
//{attribute 'qualified_only'}
VAR_GLOBAL
	
//	r_Accelerator_Setpoint	: REAL := 1E-12; (*unrealistic setpoint currently*)
	{attribute 'pytmc' := 'pv: TMO:FEE:VAC:OVRDON'}
	xSystemOverrideMode_FEE	: BOOL := FALSE; (* Global system override for the TMO FEE Vacuum System *)
	
	{attribute 'pytmc' := 'pv: TMO:NEH:VAC:OVRDON'}
	xSystemOverrideMode_TMO	: BOOL := FALSE; (* Global system override for the TMO hutch Vacuum System *)
	
	{attribute 'pytmc' := 'pv: TMO:NEH:TURBO:FAULT'}
	xTurboFault: BOOL := FALSE; (* True if any hutch turbo is not at speed or fault *)	
	
	{attribute 'pytmc' := 'pv: TMO:NEH:VALVE:FAULT'}
	xValveFault: BOOL := FALSE; (* True if any hutch turbo is not at speed or fault *)	
	
		{attribute 'pytmc' := 'pv: TMO:NEH:ALL:GCC:ENABLE'}
	xGCC_Enable_SW: BOOL := FALSE; (* True if any hutch turbo is not at speed or fault *)	
END_VAR

// ---- POUs/MAIN.TcPOU
PROGRAM MAIN
VAR

	fbLogHandler : FB_LogHandler;
	
END_VAR


fbLogHandler();

// Run the Diagnostics PRG
//DIAGNOSTICS();

(* FEE devices*)
//PRG_FEE();
PRG_Hutch_Gauges();
PRG_Hutch_Beamline_Valves();
PRG_Roughing_Pumps();

PMPS();

END_PROGRAM

// ---- POUs/PRG_Hutch_Gauges.TcPOU
PROGRAM PRG_Hutch_Gauges
VAR
END_VAR

(* Roughing Gauges *)
	TMO_ROUGH1_GPI_01.M_SetBits(32767);
	TMO_ROUGH1_GPI_01(PG=>);

	TMO_ROUGH1_GPI_02.M_SetBits(32767);
	TMO_ROUGH1_GPI_02(PG=>);

	TMO_ROUGH1_GPI_03.M_SetBits(32767);
	TMO_ROUGH1_GPI_03(PG=>);

	TMO_ROUGH2_GPI_01.M_SetBits(32767);
	TMO_ROUGH2_GPI_01(PG=>);
	
	TMO_ROUGH2_GPI_02.M_SetBits(32767);
	TMO_ROUGH2_GPI_02(PG=>);
	
	


(* Beamline Pirani & Cold Cathode*)
	MR2K4_KBO_GPI_01.M_SetBits(30518);
	MR2K4_KBO_GPI_01(); 
	
	MR2K4_KBO_GCC_01.M_SetBits(30518);
	MR2K4_KBO_GCC_01(PG:=MR2K4_KBO_GPI_01.PG , IG=> );

	PA1K4_IP1_GPI_01.M_SetBits(30518);	
	PA1K4_IP1_GPI_01(); 

	PA1K4_IP1_GCC_01.M_SetBits(30518);
	PA1K4_IP1_GCC_01(PG:=PA1K4_IP1_GPI_01.PG , IG=> );

	IM4K4_PPM_GCC_01.M_SetBits(30518);	
	IM4K4_PPM_GCC_01(PG:=PA1K4_IP1_GPI_01.PG , IG=> );

	LI2K4_IP1_GFS_01(PG:=PA1K4_IP1_GPI_01.PG , IG=> );
	
	TM1K4_GCC_01.M_SetBits(30518);
	TM1K4_GCC_01(PG:=TMO_ROUGH1_GPI_03.PG , IG=> );


	IM5K4_PPM_GCC_01.M_SetBits(30518);	
	IM5K4_PPM_GCC_01(PG:=PA2K4_IP1_GPI_01.PG , IG=> );
	
	PA2K4_IP1_GPI_01.M_SetBits(30518);
	PA2K4_IP1_GPI_01();
	
	PA2K4_IP1_GCC_01.M_SetBits(30518);
	PA2K4_IP1_GCC_01(PG:=PA2K4_IP1_GPI_01.PG , IG=> );

	MR4K4_KBO_GPI_01.M_SetBits(30518);	
	MR4K4_KBO_GPI_01();
	
	MR4K4_KBO_GCC_01.M_SetBits(30518);	
	MR4K4_KBO_GCC_01(PG:=MR4K4_KBO_GPI_01.PG , IG=> );
	

(* Auto switch on cold cathode gauges if interlock permits *)

(*
MR2K4_KBO_GCC_01.M_HVE(TRUE);
PA1K4_IP1_GCC_01.M_HVE(TRUE);
IM4K4_PPM_GCC_01.M_HVE(TRUE);
TM1K4_GCC_01.M_HVE(TRUE);
IM5K4_PPM_GCC_01.M_HVE(TRUE);
PA2K4_IP1_GCC_01.M_HVE(TRUE);
// MR4K4_KBO_GCC_01.M_HVE(TRUE);

*)

END_PROGRAM

// ---- POUs/PRG_Hutch_Beamline_Valves.TcPOU
PROGRAM PRG_Hutch_Beamline_Valves
VAR
	LAMP_C2_GCC_01: FB_MKS500; // wrong. only need temporary before integrate with LAMP 
	xAll_Turbo_isRunning : BOOL := False;
	xTurbos_are_Atspd : BOOL := False;
	xValves_are_OPN_OK : BOOL := False;
	
	ton_PA1K4_IP1_PTM_01_notRunning : TON;
	ton_PA1K4_IP1_PTM_02_notRunning : TON;
	ton_PA1K4_IP1_PTM_03_notRunning : TON;
	ton_IM4K4_PPM_PTM_01_notRunning : TON;
	ton_LI1K4_IP1_PTM_01_notRunning : TON;
	ton_LI3K4_IP1_OUT_PTM_01_notRunning : TON;
	ton_TM1K4_PTM_01_notRunning : TON;
	ton_IM5K4_PPM_PTM_01_notRunning : TON;
	
	tDelOK	:	TIME := T#30S;
	xExtIlkOK : BOOL;

	PA1K4_IP1_PTM_01_isRunning: BOOL;
	PA1K4_IP1_PTM_02_isRunning: BOOL;
	PA1K4_IP1_PTM_03_isRunning: BOOL;
	IM4K4_PPM_PTM_01_isRunning: BOOL;
	LI1K4_IP1_PTM_01_isRunning: BOOL;
	LI3K4_IP1_OUT_PTM_01_isRunning: BOOL;
	TM1K4_PTM_01_isRunning: BOOL;
	IM5K4_PPM_PTM_01_isRunning: BOOL;
	
END_VAR


(* Beamline window valves use VGC function. Valves allow to open when both upstream and downstream gauges
    reading pressure below than setpoints,  all turbo pumps are running and no faults, and all beamline valves
    in hutch are OPN_OK*)

(* check turbo pump status	*)
PA1K4_IP1_PTM_01_isRunning := PA1K4_IP1_PTM_01.iq_stPTM.eState = E_PumpState.pumpRUNNING;
ton_PA1K4_IP1_PTM_01_notRunning(IN:= NOT PA1K4_IP1_PTM_01_isRunning, PT:=tDelOK);

PA1K4_IP1_PTM_02_isRunning := PA1K4_IP1_PTM_02.iq_stPTM.eState = E_PumpState.pumpRUNNING;
ton_PA1K4_IP1_PTM_02_notRunning(IN:= NOT PA1K4_IP1_PTM_02_isRunning, PT:=tDelOK);

PA1K4_IP1_PTM_03_isRunning := PA1K4_IP1_PTM_03.iq_stPTM.eState = E_PumpState.pumpRUNNING;
ton_PA1K4_IP1_PTM_03_notRunning(IN:= NOT PA1K4_IP1_PTM_03_isRunning, PT:=tDelOK);

IM4K4_PPM_PTM_01_isRunning := IM4K4_PPM_PTM_01.iq_stPTM.eState = E_PumpState.pumpRUNNING;
ton_IM4K4_PPM_PTM_01_notRunning(IN:= NOT IM4K4_PPM_PTM_01_isRunning, PT:=tDelOK);

LI1K4_IP1_PTM_01_isRunning := LI1K4_IP1_PTM_01.iq_stPTM.eState = E_PumpState.pumpRUNNING;
ton_LI1K4_IP1_PTM_01_notRunning(IN:= NOT LI1K4_IP1_PTM_01_isRunning, PT:=tDelOK);

LI3K4_IP1_OUT_PTM_01_isRunning := LI3K4_IP1_OUT_PTM_01.iq_stPTM.eState = E_PumpState.pumpRUNNING;
ton_LI3K4_IP1_OUT_PTM_01_notRunning(IN:= NOT LI3K4_IP1_OUT_PTM_01_isRunning, PT:=tDelOK);

TM1K4_PTM_01_isRunning := TM1K4_PTM_01.iq_stPTM.eState = E_PumpState.pumpRUNNING;
ton_TM1K4_PTM_01_notRunning(IN:= NOT TM1K4_PTM_01_isRunning, PT:=tDelOK);

IM5K4_PPM_PTM_01_isRunning := IM5K4_PPM_PTM_01.iq_stPTM.eState = E_PumpState.pumpRUNNING;
ton_IM5K4_PPM_PTM_01_notRunning(IN:= NOT IM5K4_PPM_PTM_01_isRunning, PT:=tDelOK);

xTurboFault := ton_PA1K4_IP1_PTM_01_notRunning.Q OR ton_PA1K4_IP1_PTM_02_notRunning.Q OR
               ton_PA1K4_IP1_PTM_03_notRunning.Q OR ton_IM4K4_PPM_PTM_01_notRunning.Q OR
			   ton_LI1K4_IP1_PTM_01_notRunning.Q OR ton_LI3K4_IP1_OUT_PTM_01_notRunning.Q OR
				ton_TM1K4_PTM_01_notRunning.Q OR ton_IM5K4_PPM_PTM_01_notRunning.Q ;

(* check beamline valve OPEN permit *)	
xValves_are_OPN_OK :=  MR2K4_KBO_VWC_01.iq_stValve.xOPN_OK AND MR3K4_KBO_VWC_01.iq_stValve.xOPN_OK AND
                       LI3K4_IP1_VWC_01.iq_stValve.xOPN_OK AND PC5K4_VWC_01.iq_stValve.xOPN_OK ;  

(*set xValveFault to True, if not all beamline valves are OPN_OK*)
IF NOT xValves_are_OPN_OK Then
	xValveFault := TRUE;
ElSE
   xValveFault := False;	
END_IF
					   
   
					 

MR2K4_KBO_VWC_01(
				i_stUSG := MR2K4_KBO_GCC_01.IG, 
				i_stDSG:= MR2K4_KBO_GCC_01.IG, 
				i_xDis_DPIlk := FALSE, 
				i_xEPS_OK := TRUE,
				i_xPMPS_OK := TRUE, 
				i_xExt_OK := NOT xTurboFault AND xValves_are_OPN_OK, 
				i_xOverrideMode := xSystemOverrideMode_TMO, 
				i_xReset := xReset_PMPS_FFO2,
				io_fbFFHWO :=g_FastFaultOutput2,
                fbArbiter := g_fbArbiter1,
				
);


MR3K4_KBO_VWC_01(
				i_stUSG := MR2K4_KBO_GCC_01.IG, 
				i_stDSG:= PA1K4_IP1_GCC_01.IG, 
				i_xDis_DPIlk := FALSE, 
				i_xEPS_OK := TRUE,
				i_xPMPS_OK := TRUE, 
				i_xExt_OK := xTurbos_are_Atspd AND xValves_are_OPN_OK, 
				i_xOverrideMode := xSystemOverrideMode_TMO, 
				i_xReset := xReset_PMPS_FFO2,
				io_fbFFHWO :=g_FastFaultOutput2,
                fbArbiter := g_fbArbiter1);

LI3K4_IP1_VWC_01(
				i_stUSG := LAMP_C2_GCC_01.IG, 
				i_stDSG:= IM5K4_PPM_GCC_01.IG, 
				i_xDis_DPIlk := FALSE, 
				i_xEPS_OK := TRUE,
				i_xPMPS_OK := TRUE, 
				i_xExt_OK := xTurbos_are_Atspd AND xValves_are_OPN_OK, 
				i_xOverrideMode := xSystemOverrideMode_TMO,
				i_xReset := xReset_PMPS_FFO2,
				io_fbFFHWO :=g_FastFaultOutput2,
                fbArbiter := g_fbArbiter1);

PC5K4_VWC_01(
				i_stUSG := IM5K4_PPM_GCC_01.IG, 
				i_stDSG:= PA2K4_IP1_GCC_01.IG, 
				i_xDis_DPIlk := FALSE, 
				i_xEPS_OK := TRUE,
				i_xPMPS_OK := TRUE, 
				i_xExt_OK := xTurbos_are_Atspd AND xValves_are_OPN_OK, 
				i_xOverrideMode := xSystemOverrideMode_TMO, 
				i_xReset := xReset_PMPS_FFO2,
				io_fbFFHWO :=g_FastFaultOutput2,
                fbArbiter := g_fbArbiter1);

(* MR4K4_KBO_VWC_01(
				i_stUSG := PA2K4_IP1_GCC_01.IG, 
				i_stDSG:= MR4K4_KBO_GCC_01.IG, 
				i_xDis_DPIlk := FALSE, 
				i_xEPS_OK := TRUE,
				i_xPMPS_OK := TRUE, 
				i_xExt_OK := xTurbos_are_Atspd AND xValves_are_OPN_OK, 
				i_xOverrideMode := xSystemOverrideMode_TMO, 
				i_xReset := xReset_PMPS_FFO2,
				io_fbFFHWO :=g_FastFaultOutput2,
                fbArbiter := g_fbArbiter1);
	
*)

END_PROGRAM

// ---- POUs/PRG_Roughing_Pumps.TcPOU
PROGRAM PRG_Roughing_Pumps
VAR
	
	xRough1Vrc01_OpenOK: BOOL := False;
	xRough1Vrc02_OpenOK: BOOL := False;
	xRough2Vrc01_OpenOK: BOOL := False;
	dummy_FFFO : FB_HardwareFFOutput;
	dummy_fbArbiter1    :   FB_Arbiter(1);
	
	PA1K4_IP1_PTM_01_xExtIlkOK: BOOL := FALSE;
	PA1K4_IP1_PTM_02_xExtIlkOK: BOOL := FALSE;
	PA1K4_IP1_PTM_03_xExtIlkOK: BOOL := False;
	
	

	tonDelOK : TON;
	tDelOK	:	TIME := T#30S;
	xExtIlkOK : BOOL;
	
	
	
	
	IM4K4_PPM_PTM_01_xExtIlkOK: BOOL := FALSE;
	LI1K4_IP1_PTM_01_xExtIlkOK: BOOL := FALSE;
	LI3K4_IP1_OUT_PTM_01_xExtIlkOK: BOOL := False;
	IM5K4_PPM_PTM_01_xExtIlkOK: BOOL := False;
	
	rTolerance : REAL;
	xDifPressureOK : BOOL := FALSE;
	TMO_ROUGH1_VRC_01_xExt_OK : BOOL;
	TMO_ROUGH1_VRC_02_xExt_OK : BOOL;
	
END_VAR

VAR RETAIN
	TM1K4_PTM_01_xExtIlkOK: BOOL := False;
END_VAR


(* Roughing Valves *)

(* All three roughing valves permit to open when both side reading pressure below than setpoint, 1E-3 for both sides.
   When chamber is vented, bypass to open valve to pump down. 
   FB_VGC_2S is used for VRC controls.
   
   For TMO_ROUGH1_VRC_01 & TMO_ROUGH1_VRC_02, additional interlock is implemented using i_xExt_OK input of VGC function:
   If pressure difference between TMO_ROUGH1_GPI_02 and TMO_ROUGH1_GPI_03 is greater than 20 Torr, 
   only one of them permit to open.
   
*)


(* Check the pressure difference between TMO_ROUGH1_GPI_02 and TMO_ROUGH1_GPI_03 *) 



rTolerance := 0.1;
xDifPressureOK := (ABS(TMO_ROUGH1_GPI_02.PG.rPRESS - TMO_ROUGH1_GPI_03.PG.rPRESS ) <= rTolerance ) AND
				  TMO_ROUGH1_GPI_02.PG.xPRESS_OK AND TMO_ROUGH1_GPI_03.PG.xPRESS_OK;
				  
(* Set external interlock OK TRUE, when xDifPressureOK or TMO_ROUGH1_VRC_02 is closed *)				  
TMO_ROUGH1_VRC_01_xExt_OK := xDifPressureOK OR TMO_ROUGH1_VRC_02.iq_stValve.i_xClsLS; 
TMO_ROUGH1_VRC_02_xExt_OK := xDifPressureOK OR TMO_ROUGH1_VRC_01.iq_stValve.i_xClsLS; 


TMO_ROUGH1_VRC_01(
				i_stUSG := TMO_ROUGH1_GPI_02.PG, 
				i_stDSG:= TMO_ROUGH1_GPI_01.PG, 
				i_xDis_DPIlk := FALSE, 
				i_xEPS_OK := TRUE,
				i_xPMPS_OK := TRUE, 
				i_xExt_OK := TMO_ROUGH1_VRC_01_xExt_OK, 
				i_xOverrideMode := xSystemOverrideMode_TMO AND TMO_ROUGH1_VRC_01_xExt_OK,
				i_xReset := False,
				io_fbFFHWO :=dummy_FFFO,
                fbArbiter := dummy_fbArbiter1,
);


TMO_ROUGH1_VRC_02(
				i_stUSG := TMO_ROUGH1_GPI_03.PG, 
				i_stDSG:= TMO_ROUGH1_GPI_01.PG, 
				i_xDis_DPIlk := FALSE, 
				i_xEPS_OK := TRUE,
				i_xPMPS_OK := TRUE, 
				i_xExt_OK := TMO_ROUGH1_VRC_02_xExt_OK, 
				i_xOverrideMode := xSystemOverrideMode_TMO AND TMO_ROUGH1_VRC_02_xExt_OK, 
				i_xReset := false,
				io_fbFFHWO :=dummy_FFFO,
                fbArbiter := dummy_fbArbiter1);


TMO_ROUGH2_VRC_01(
				i_stUSG := TMO_ROUGH2_GPI_02.PG, 
				i_stDSG:= TMO_ROUGH2_GPI_01.PG, 
				i_xDis_DPIlk := FALSE, 
				i_xEPS_OK := TRUE,
				i_xPMPS_OK := TRUE, 
				i_xExt_OK := TRUE, 
				i_xOverrideMode := xSystemOverrideMode_TMO, 
				i_xReset := false,
				io_fbFFHWO :=dummy_FFFO,
                fbArbiter := dummy_fbArbiter1);


(* Granite 1 K4S2 Differential Turbo pumps *)


(* check if PA1K4_IP1_PTM_03 is Atspd, if it is starting, set up a timer for 30s to *)

xExtIlkOK := F_Turbo_Protection_ILK(i_stTurbo := PA1K4_IP1_PTM_01.iq_stPTM, 
			i_stISG := PA1K4_IP1_GPI_01.PG, 
			i_stBSG := TMO_ROUGH1_GPI_02.PG, 
			iq_stValve := TMO_ROUGH1_VRC_01.iq_stValve)	;
					
(* delay 30s to start if PTM03 is not at speed*)
IF (PA1K4_IP1_PTM_03.iq_stPTM.i_xAtSpd) AND (NOT PA1K4_IP1_PTM_03.iq_stPTM.i_xFault) THEN
		PA1K4_IP1_PTM_01_xExtIlkOK := xExtIlkOK;

ELSIF (PA1K4_IP1_PTM_03.iq_stPTM.q_RunDO ) AND (NOT PA1K4_IP1_PTM_03.iq_stPTM.i_xFault ) THEN
	//delay timer
  	  tonDelOK(IN:= xExtIlkOK, PT:=tDelOK);
	PA1K4_IP1_PTM_01_xExtIlkOK := xExtIlkOK AND tonDelOK.Q;	
ELSE
		PA1K4_IP1_PTM_01_xExtIlkOK := FALSE;			
END_IF


xExtIlkOK := F_Turbo_Protection_ILK(i_stTurbo := PA1K4_IP1_PTM_02.iq_stPTM, 
			i_stISG := PA1K4_IP1_GPI_01.PG, 
			i_stBSG := TMO_ROUGH1_GPI_02.PG, 
			iq_stValve := TMO_ROUGH1_VRC_01.iq_stValve)	;

IF (PA1K4_IP1_PTM_03.iq_stPTM.i_xAtSpd) AND (NOT PA1K4_IP1_PTM_03.iq_stPTM.i_xFault) THEN
		PA1K4_IP1_PTM_02_xExtIlkOK := xExtIlkOK;

ELSIF (PA1K4_IP1_PTM_03.iq_stPTM.q_RunDO ) AND (NOT PA1K4_IP1_PTM_03.iq_stPTM.i_xFault ) THEN
	//delay timer
  	  tonDelOK(IN:= xExtIlkOK, PT:=tDelOK);
	PA1K4_IP1_PTM_02_xExtIlkOK := xExtIlkOK AND tonDelOK.Q;	
ELSE
		PA1K4_IP1_PTM_02_xExtIlkOK := FALSE;			
END_IF

PA1K4_IP1_PTM_03_xExtIlkOK  := F_Turbo_Protection_ILK(i_stTurbo := PA1K4_IP1_PTM_03.iq_stPTM, 
			i_stISG := PA1K4_IP1_GPI_01.PG, 
			i_stBSG := TMO_ROUGH1_GPI_02.PG, 
			iq_stValve := TMO_ROUGH1_VRC_01.iq_stValve)	;


PA1K4_IP1_PTM_01(i_xExtIlkOK := PA1K4_IP1_PTM_01_xExtIlkOK , iq_stPTM => );

PA1K4_IP1_PTM_02(i_xExtIlkOK := PA1K4_IP1_PTM_02_xExtIlkOK, iq_stPTM => );
PA1K4_IP1_PTM_03(i_xExtIlkOK := PA1K4_IP1_PTM_03_xExtIlkOK, iq_stPTM => );

(*Serial Interface*)
(*Assign adresses to the pfeiffer controllers connected to this serial terminal*)
st_Pfeiffer_CTRL_PTM_01_02_03[1].iSerialAddress :=10;//PA1K4_IP1_PTM_01
st_Pfeiffer_CTRL_PTM_01_02_03[1].xEnableComm := TRUE;
st_Pfeiffer_CTRL_PTM_01_02_03[2].iSerialAddress :=9;//PA1K4_IP1_PTM_02
st_Pfeiffer_CTRL_PTM_01_02_03[2].xEnableComm := TRUE;
st_Pfeiffer_CTRL_PTM_01_02_03[3].iSerialAddress :=18;//PA1K4_IP1_PTM_03
st_Pfeiffer_CTRL_PTM_01_02_03[3].xEnableComm := TRUE;	
(* Instanitate the Function block for serial communication with Pfeiffer*)	
PA1K4_IP1_PTM_01_02_03_COM(astPfeifferControl := st_Pfeiffer_CTRL_PTM_01_02_03,
			   astPfeifferStatus:= st_Pfeiffer_RBK_PTM_01_02_03,
				SerialRXBuffer:= K4S2_02_E10_SerialRXBuffer,
				SerialTXBuffer:= K4S2_02_E10_SerialTXBuffer);
(* Copy Status Pv's into the PTM structure*)
PA1K4_IP1_PTM_01.M_Serial_IO(st_Pfeiffer_CTRL=>st_Pfeiffer_CTRL_PTM_01_02_03[1],st_Pfeiffer_RBK:=st_Pfeiffer_RBK_PTM_01_02_03[1]);				
PA1K4_IP1_PTM_02.M_Serial_IO(st_Pfeiffer_CTRL=>st_Pfeiffer_CTRL_PTM_01_02_03[2],st_Pfeiffer_RBK:=st_Pfeiffer_RBK_PTM_01_02_03[2]);				
PA1K4_IP1_PTM_03.M_Serial_IO(st_Pfeiffer_CTRL=>st_Pfeiffer_CTRL_PTM_01_02_03[3],st_Pfeiffer_RBK:=st_Pfeiffer_RBK_PTM_01_02_03[3]);				
		
(* Leybold turbo pumps on Granite 1 *)

IM4K4_PPM_PTM_01_xExtIlkOK := F_Turbo_Protection_ILK(i_stTurbo := IM4K4_PPM_PTM_01.iq_stPTM, 
			i_stISG := PA1K4_IP1_GPI_01.PG, 
			i_stBSG := TMO_ROUGH1_GPI_02.PG, 
			iq_stValve := TMO_ROUGH1_VRC_01.iq_stValve)	;

IM4K4_PPM_PTM_01(i_xExtIlkOK := IM4K4_PPM_PTM_01_xExtIlkOK, iq_stPTM => );

(* Instanitate the Function block for serial communication with TD20 *)
IM4K4_PPM_PTM_01_COM(SerialRXBuffer := K4S2_02_E17_SerialRXBuffer, 
				SerialTXBuffer:= K4S2_02_E17_SerialTXBuffer,
				astTD20Status=>);
(* Copy Status Pv's into the PTM structure*)
IM4K4_PPM_PTM_01.M_Serial_IO(IM4K4_PPM_PTM_01_COM.astTD20Status);



LI1K4_IP1_PTM_01_xExtIlkOK := F_Turbo_Protection_ILK(i_stTurbo := LI1K4_IP1_PTM_01.iq_stPTM, 
			i_stISG := PA1K4_IP1_GPI_01.PG, 
			i_stBSG := TMO_ROUGH1_GPI_02.PG, 
			iq_stValve := TMO_ROUGH1_VRC_01.iq_stValve)	;
			
LI1K4_IP1_PTM_01(i_xExtIlkOK := LI1K4_IP1_PTM_01_xExtIlkOK, iq_stPTM => );

(* Instanitate the Function block for serial communication with TD20 *)
LI1K4_IP1_PTM_01_COM(SerialRXBuffer := K4S2_02_E18_SerialRXBuffer, 
				SerialTXBuffer:= K4S2_02_E18_SerialTXBuffer,
				astTD20Status=>);
(* Copy Status Pv's into the PTM structure*)
LI1K4_IP1_PTM_01.M_Serial_IO(LI1K4_IP1_PTM_01_COM.astTD20Status);



(* Granite 2 K4S6 *)

LI3K4_IP1_OUT_PTM_01_xExtIlkOK := F_Turbo_Protection_ILK(i_stTurbo := LI3K4_IP1_OUT_PTM_01.iq_stPTM, 
			i_stISG := PA2K4_IP1_GPI_01.PG, 
			i_stBSG := TMO_ROUGH1_GPI_03.PG, 
			iq_stValve := TMO_ROUGH1_VRC_02.iq_stValve)	;

LI3K4_IP1_OUT_PTM_01(i_xExtIlkOK := LI3K4_IP1_OUT_PTM_01_xExtIlkOK, iq_stPTM => );

TM1K4_PTM_01_xExtIlkOK := F_Turbo_Protection_ILK(i_stTurbo := TM1K4_PTM_01.iq_stPTM, 
			i_stISG := PA2K4_IP1_GPI_01.PG, 
			i_stBSG := TMO_ROUGH1_GPI_03.PG, 
			iq_stValve := TMO_ROUGH1_VRC_02.iq_stValve)	;

TM1K4_PTM_01(i_xExtIlkOK := TM1K4_PTM_01_xExtIlkOK, iq_stPTM => );

IM5K4_PPM_PTM_01_xExtIlkOK := F_Turbo_Protection_ILK(i_stTurbo := IM5K4_PPM_PTM_01.iq_stPTM, 
			i_stISG := PA2K4_IP1_GPI_01.PG, 
			i_stBSG := TMO_ROUGH1_GPI_03.PG, 
			iq_stValve := TMO_ROUGH1_VRC_02.iq_stValve)	;
			
IM5K4_PPM_PTM_01(i_xExtIlkOK := IM5K4_PPM_PTM_01_xExtIlkOK, iq_stPTM => );

(*Serial Interface*)
(*Assign adresses to the pfeiffer controllers connected to this serial terminal*)
st_Pfeiffer_CTRL_PTM_Granite2[1].iSerialAddress :=1;//LI3K4_IP1_OUT_PTM_01
st_Pfeiffer_CTRL_PTM_Granite2[1].xEnableComm := TRUE;
st_Pfeiffer_CTRL_PTM_Granite2[2].iSerialAddress :=7;//TM1K4_PTM_01
st_Pfeiffer_CTRL_PTM_Granite2[2].xEnableComm := TRUE;
st_Pfeiffer_CTRL_PTM_Granite2[3].iSerialAddress :=9; //IM5K4_PPM_PTM_01
st_Pfeiffer_CTRL_PTM_Granite2[3].xEnableComm := TRUE;	
(* Instanitate the Function block for serial communication with Pfeiffer*)	
Granite2_PTM_COM(astPfeifferControl := st_Pfeiffer_CTRL_PTM_Granite2,
			   astPfeifferStatus:= st_Pfeiffer_RBK_PTM_Granite2,
				SerialRXBuffer:= K4S6_01_E5_SerialRXBuffer,
				SerialTXBuffer:= K4S6_01_E5_SerialTXBuffer);
(* Copy Status Pv's into the PTM structure*)
LI3K4_IP1_OUT_PTM_01.M_Serial_IO(st_Pfeiffer_CTRL=>st_Pfeiffer_CTRL_PTM_Granite2[1],st_Pfeiffer_RBK:=st_Pfeiffer_RBK_PTM_Granite2[1]);				
TM1K4_PTM_01.M_Serial_IO(st_Pfeiffer_CTRL=>st_Pfeiffer_CTRL_PTM_Granite2[2],st_Pfeiffer_RBK:=st_Pfeiffer_RBK_PTM_Granite2[2]);				
IM5K4_PPM_PTM_01.M_Serial_IO(st_Pfeiffer_CTRL=>st_Pfeiffer_CTRL_PTM_Granite2[3],st_Pfeiffer_RBK:=st_Pfeiffer_RBK_PTM_Granite2[3]);

END_PROGRAM

// ---- POUs/F_Turbo_Protection_ILK.TcPOU
FUNCTION F_Turbo_Protection_ILK : BOOL
VAR_INPUT
	i_Turbo : ST_PTM; // Turbo Pump
	i_stISG : ST_VG; //Gauge measuring inlet Pressure e.g Pirani
	i_stBSG : ST_VG; //Gauge measureing backing pressure
	iq_stValve : ST_VRC; //
END_VAR
VAR
END_VAR


F_Turbo_Protection_ILK := (i_stISG.xPRESS_OK AND i_stISG.rPRESS < i_Turbo.rInletPressureSP) AND (i_stBSG.xPRESS_OK AND i_stBSG.rPRESS < i_Turbo.rBackingPressureSP)AND iq_stValve.i_xOpnLS;

END_FUNCTION

// ---- POUs/PRG_FEE.TcPOU
 PROGRAM PRG_FEE
VAR
ADS_connection_counter : UDINT;	

(*Upstream Interface*)
	
    USG_PIP : ST_VG;
	
	USG_VGC : ST_VG;


END_VAR

(* Gauges*)
   (* Read GCC from upstream PLC - plc-kfe-vac*)
  (* MR1K4_GCC_01_ADS(
	sNetId:= '172.21.92.61.1.1', 
	nPort:=851 , 
	sVarName:= 'fb_MR1K4_SOMS_GCC_1' , 
	iWatchdog:=ADS_connection_counter , 
	IG=> , 
	bError=> ); *)
	(* if upstream vacuum ok, set upstream press at good levels *)  
    IF USVacOk_HI THEN 
		USG_VGC.xAT_VAC := TRUE;
		USG_VGC.rPRESS := 5E-7;
		USG_VGC.xPRESS_OK := TRUE;
	ELSE
		USG_VGC.xPRESS_OK := FALSE;
		USG_VGC.xAT_VAC := FALSE;
	END_IF

    IF USVacOk_LO THEN 
		USG_PIP.rPRESS := 5E-5;
		USG_PIP.xPRESS_OK := TRUE;
		USG_PIP.xAT_VAC := TRUE;
	ELSE
		USG_PIP.xPRESS_OK := FALSE;
		USG_PIP.xAT_VAC := FALSE;
	END_IF 

	(* check other gauges*)
	TV1K4_GPI_01(); 
	ST1K4_TEST_GPI_01(); 
	ST2K4_BCS_GPI_01();
	PC4K4_XTES_GPI_01(); 
	
	TV1k4_GCC_01(PG:=TV1k4_GPI_01.PG , IG=> , bEP := TRUE);
	ST1K4_TEST_GCC_01(PG:=ST1K4_TEST_GPI_01.PG , IG=>, bEP := TRUE ); 
	ST2K4_BCS_GCC_01(PG:=ST2K4_BCS_GPI_01.PG , IG=>, bEP := TRUE );
	PC4K4_XTES_GCC_01(PG:=PC4K4_XTES_GPI_01.PG , IG=>, bEP := TRUE );
		
(* Valves*)
(*example
GEM1_VGC_10(i_stUSG := USG_GCC.IG, i_stDSG:= GEM1_GCC_10.IG,i_xDis_DPIlk := TRUE, i_xEPS_OK := TRUE,
		i_xPMPS_OK := TRUE, i_xExt_OK := xGEM1_AperturesOpnOK, i_xOverrideMode := xGEM1OverrideMode,i_xReset := xFastFaultReset,io_fbFFHWO :=g_FastFaultOutput1);
*)
	TV1K4_VGC_01(
				i_stUSG := USG_VGC, 
				i_stDSG:= TV1k4_GCC_01.IG, 
				i_xDis_DPIlk := FALSE, 
				i_xEPS_OK := TRUE,
				i_xPMPS_OK := TRUE, 
				i_xExt_OK := TRUE, 
				i_xOverrideMode := xSystemOverrideMode_FEE, 
				i_xReset := xReset_PMPS_FFO1,
				io_fbFFHWO :=g_FastFaultOutput1,
				fbArbiter := g_fbArbiter1);
	
 	TV1K4_VGC_02(
				i_stUSG := TV1k4_GCC_01.IG, 
				i_stDSG:= ST1K4_TEST_GCC_01.IG, 
				i_xDis_DPIlk := FALSE, 
				i_xEPS_OK := TRUE,
				i_xPMPS_OK := TRUE, 
				i_xExt_OK := TRUE, 
				i_xOverrideMode := xSystemOverrideMode_FEE, 
				i_xReset := xReset_PMPS_FFO1,
				io_fbFFHWO :=g_FastFaultOutput1,
                fbArbiter := g_fbArbiter1);
	
	ST3K4_PPS_VGC_01(
				i_stUSG := ST2K4_BCS_GCC_01.IG, 
				i_stDSG:= PC4K4_XTES_GCC_01.IG, 
				i_xDis_DPIlk := FALSE, 
				i_xEPS_OK := TRUE,
				i_xPMPS_OK := TRUE, 
				i_xExt_OK := TRUE, 
				i_xOverrideMode := xSystemOverrideMode_FEE, 
				i_xReset := xReset_PMPS_FFO2,
				io_fbFFHWO :=g_FastFaultOutput2,
                fbArbiter := g_fbArbiter1);
				
(*Ion Pumps*)	
	(*example
	SP1L0_KMONO_PIP_01(i_stGauge:=SP1L0_KMONO_GCC_01.IG, stPump=>);*)		

	MR1K4_SOMS_PIP_01(i_stGauge := USG_PIP, stPump=>);
	ST1K4_TEST_PIP_01(i_stGauge := ST1K4_TEST_GCC_01.IG, stPump=>);
	ST2K4_BCS_PIP_01(i_stGauge := ST2K4_BCS_GCC_01.IG, stPump=>);
	ST3K4_PPS_PIP_01(i_stGauge := ST2K4_BCS_GCC_01.IG, stPump=>);
	PC4K4_XTES_PIP_01(i_stGauge := PC4K4_XTES_GCC_01.IG, stPump=>);

END_PROGRAM
